LIN {X 0,Y 531.944,Z 396.877,A -85,B 0,C 180,E1 -4217.795,E2 -4217.795} C_VEL
LIN {X 0,Y 531.768,Z 407.802,A -85,B 0,C 180,E1 -4218.459,E2 -4218.459} C_VEL
LIN {X 0,Y 531.496,Z 419.072,A -85,B 0,C 180,E1 -4219.33,E2 -4219.33} C_VEL
LIN {X 0,Y 531.238,Z 429.006,A -85,B 0,C 180,E1 -4220.288,E2 -4220.288} C_VEL
LIN {X 0,Y 530.96,Z 438.48,A -85,B 0,C 180,E1 -4221.435,E2 -4221.435} C_VEL
LIN {X 0,Y 530.755,Z 446.079,A -85,B 0,C 180,E1 -4222.58,E2 -4222.58} C_VEL
LIN {X 0,Y 530.616,Z 451.92,A -85,B 0,C 180,E1 -4223.683,E2 -4223.683} C_VEL
LIN {X 0,Y 530.532,Z 456.21,A -85,B 0,C 180,E1 -4224.678,E2 -4224.678} C_VEL
LIN {X 0,Y 530.523,Z 460.056,A -85,B 0,C 180,E1 -4225.82,E2 -4225.82} C_VEL
LIN {X 0,Y 530.487,Z 462.909,A -85,B 0,C 180,E1 -4226.961,E2 -4226.961} C_VEL
LIN {X 0,Y 530.412,Z 464.34,A -85,B 0,C 180,E1 -4227.72,E2 -4227.72} C_VEL
LIN {X 0,Y 530.345,Z 465.895,A -85,B 0,C 180,E1 -4229.239,E2 -4229.239} C_VEL
LIN {X 0,Y 530.345,Z 466.145,A -85,B 0,C 180,E1 -4229.998,E2 -4229.998} C_VEL
LIN {X 0,Y 530.361,Z 465.393,A -85,B 0,C 180,E1 -4231.517,E2 -4231.517} C_VEL
LIN {X 0,Y 530.411,Z 464.474,A -85,B 0,C 180,E1 -4232.276,E2 -4232.276} C_VEL
LIN {X 0,Y 530.516,Z 461.35,A -85,B 0,C 180,E1 -4233.796,E2 -4233.796} C_VEL
LIN {X 0,Y 530.485,Z 457.917,A -85,B 0,C 180,E1 -4234.938,E2 -4234.938} C_VEL
LIN {X 0,Y 530.621,Z 453.388,A -85,B 0,C 180,E1 -4236.08,E2 -4236.08} C_VEL
LIN {X 0,Y 530.719,Z 447.667,A -85,B 0,C 180,E1 -4237.225,E2 -4237.225} C_VEL
LIN {X 0,Y 530.93,Z 440.518,A -85,B 0,C 180,E1 -4238.37,E2 -4238.37} C_VEL
LIN {X 0,Y 531.119,Z 433.212,A -85,B 0,C 180,E1 -4239.327,E2 -4239.327} C_VEL
LIN {X 0,Y 531.352,Z 423.28,A -85,B 0,C 180,E1 -4240.38,E2 -4240.38} C_VEL
LIN {X 0,Y 531.625,Z 413.173,A -85,B 0,C 180,E1 -4241.242,E2 -4241.242} C_VEL
LIN {X 0,Y 531.843,Z 401.662,A -85,B 0,C 180,E1 -4242.025,E2 -4242.025} C_VEL
LIN {X 0,Y 532.086,Z 388.922,A -85,B 0,C 180,E1 -4242.683,E2 -4242.683} C_VEL
LIN {X 0,Y 532.305,Z 376.104,A -85,B 0,C 180,E1 -4243.163,E2 -4243.163} C_VEL
LIN {X 0,Y 532.142,Z 370.063,A -85,B 0,C 180,E1 -4243.337,E2 -4243.337} C_VEL
LIN {X 0,Y 530.699,Z 362.74,A -85,B 0,C 180,E1 -4243.544,E2 -4243.544} C_VEL
LIN {X 0,Y 530.77,Z 357.319,A -85,B 0,C 180,E1 -4246.142,E2 -4246.142} C_VEL
LIN {X 0,Y 530.851,Z 352.311,A -85,B 0,C 180,E1 -4248.524,E2 -4248.524} C_VEL
LIN {X 0,Y 530.919,Z 347.179,A -85,B 0,C 180,E1 -4250.939,E2 -4250.939} C_VEL
LIN {X 0,Y 531.003,Z 340.698,A -85,B 0,C 180,E1 -4254.043,E2 -4254.043} C_VEL
LIN {X 0,Y 531.083,Z 335.26,A -85,B 0,C 180,E1 -4256.737,E2 -4256.737} C_VEL
LIN {X 0,Y 531.199,Z 330.065,A -85,B 0,C 180,E1 -4259.307,E2 -4259.307} C_VEL
LIN {X 0,Y 531.287,Z 323.918,A -85,B 0,C 180,E1 -4262.155,E2 -4262.155} C_VEL
LIN {X 0,Y 531.296,Z 317.258,A -85,B 0,C 180,E1 -4264.901,E2 -4264.901} C_VEL
LIN {X 0,Y 531.069,Z 314.65,A -85,B 0,C 180,E1 -4265.908,E2 -4265.908} C_VEL
LIN {X 0,Y 530.976,Z 314.657,A -85,B 0,C 180,E1 -4269.441,E2 -4269.441} C_VEL
LIN {X 0,Y 530.948,Z 314.659,A -85,B 0,C 180,E1 -4272.456,E2 -4272.456} C_VEL
LIN {X 0,Y 530.97,Z 314.657,A -85,B 0,C 180,E1 -4275.619,E2 -4275.619} C_VEL
LIN {X 0,Y 531.003,Z 314.656,A -85,B 0,C 180,E1 -4278.565,E2 -4278.565} C_VEL
LIN {X 0,Y 531.005,Z 314.656,A -85,B 0,C 180,E1 -4280.558,E2 -4280.558} C_VEL
LIN {X 0,Y 530.953,Z 314.663,A -85,B 0,C 180,E1 -4283.841,E2 -4283.841} C_VEL
LIN {X 0,Y 530.979,Z 314.653,A -85,B 0,C 180,E1 -4286.492,E2 -4286.492} C_VEL
LIN {X 0,Y 530.953,Z 314.66,A -85,B 0,C 180,E1 -4289.353,E2 -4289.353} C_VEL
LIN {X 0,Y 530.997,Z 314.656,A -85,B 0,C 180,E1 -4292.464,E2 -4292.464} C_VEL
LIN {X 0,Y 531,Z 314.652,A -85,B 0,C 180,E1 -4294.942,E2 -4294.942} C_VEL
LIN {X 0,Y 530.986,Z 314.657,A -85,B 0,C 180,E1 -4297.888,E2 -4297.888} C_VEL
LIN {X 0,Y 530.971,Z 314.654,A -85,B 0,C 180,E1 -4300.676,E2 -4300.676} C_VEL
LIN {X 0,Y 530.96,Z 314.662,A -85,B 0,C 180,E1 -4303.07,E2 -4303.07} C_VEL
LIN {X 0,Y 530.995,Z 314.649,A -85,B 0,C 180,E1 -4305.435,E2 -4305.435} C_VEL
LIN {X 0,Y 531.038,Z 314.65,A -85,B 0,C 180,E1 -4308.549,E2 -4308.549} C_VEL
LIN {X 0,Y 531.04,Z 314.647,A -85,B 0,C 180,E1 -4311.629,E2 -4311.629} C_VEL
LIN {X 0,Y 531.118,Z 314.635,A -85,B 0,C 180,E1 -4314.685,E2 -4314.685} C_VEL
LIN {X 0,Y 531.105,Z 314.639,A -85,B 0,C 180,E1 -4317.725,E2 -4317.725} C_VEL
LIN {X 0,Y 531.135,Z 314.637,A -85,B 0,C 180,E1 -4320.758,E2 -4320.758} C_VEL
LIN {X 0,Y 531.092,Z 314.64,A -85,B 0,C 180,E1 -4323.034,E2 -4323.034} C_VEL
LIN {X 0,Y 531.072,Z 314.646,A -85,B 0,C 180,E1 -4326.077,E2 -4326.077} C_VEL
LIN {X 0,Y 531.015,Z 314.654,A -85,B 0,C 180,E1 -4329.138,E2 -4329.138} C_VEL
LIN {X 0,Y 531.041,Z 314.647,A -85,B 0,C 180,E1 -4331.681,E2 -4331.681} C_VEL
LIN {X 0,Y 531.004,Z 314.653,A -85,B 0,C 180,E1 -4334.956,E2 -4334.956} C_VEL
LIN {X 0,Y 531.005,Z 314.653,A -85,B 0,C 180,E1 -4337.722,E2 -4337.722} C_VEL
LIN {X 0,Y 530.985,Z 314.654,A -85,B 0,C 180,E1 -4340.938,E2 -4340.938} C_VEL
LIN {X 0,Y 530.993,Z 314.652,A -85,B 0,C 180,E1 -4344.048,E2 -4344.048} C_VEL
LIN {X 0,Y 530.971,Z 314.66,A -85,B 0,C 180,E1 -4346.745,E2 -4346.745} C_VEL
LIN {X 0,Y 530.958,Z 314.656,A -85,B 0,C 180,E1 -4349.324,E2 -4349.324} C_VEL
LIN {X 0,Y 530.959,Z 314.663,A -85,B 0,C 180,E1 -4352.105,E2 -4352.105} C_VEL
LIN {X 0,Y 530.972,Z 314.656,A -85,B 0,C 180,E1 -4354.856,E2 -4354.856} C_VEL
LIN {X 0,Y 530.953,Z 314.661,A -85,B 0,C 180,E1 -4357.508,E2 -4357.508} C_VEL
LIN {X 0,Y 530.964,Z 314.658,A -85,B 0,C 180,E1 -4360.434,E2 -4360.434} C_VEL
LIN {X 0,Y 530.94,Z 314.658,A -85,B 0,C 180,E1 -4363.283,E2 -4363.283} C_VEL
LIN {X 0,Y 530.969,Z 314.659,A -85,B 0,C 180,E1 -4365.623,E2 -4365.623} C_VEL
LIN {X 0,Y 531.002,Z 314.655,A -85,B 0,C 180,E1 -4368.569,E2 -4368.569} C_VEL
LIN {X 0,Y 530.962,Z 314.677,A -85,B 0,C 180,E1 -4370.946,E2 -4370.946} C_VEL
LIN {X 0,Y 534.217,Z 325.862,A -85,B 0,C 180,E1 -4373.111,E2 -4373.111} C_VEL
LIN {X 0,Y 536.261,Z 334.019,A -85,B 0,C 180,E1 -4374.572,E2 -4374.572} C_VEL
LIN {X 0,Y 535.432,Z 353.193,A -85,B 0,C 180,E1 -4377.445,E2 -4377.445} C_VEL
LIN {X 0,Y 534.6,Z 374.419,A -85,B 0,C 180,E1 -4380.536,E2 -4380.536} C_VEL
LIN {X 0,Y 533.898,Z 393.207,A -85,B 0,C 180,E1 -4383.204,E2 -4383.204} C_VEL
LIN {X 0,Y 533.249,Z 412.473,A -85,B 0,C 180,E1 -4385.888,E2 -4385.888} C_VEL
LIN {X 0,Y 533.044,Z 420.982,A -85,B 0,C 180,E1 -4387.036,E2 -4387.036} C_VEL
LIN {X 0,Y 536.002,Z 434.729,A -85,B 0,C 180,E1 -4387.369,E2 -4387.369} C_VEL
LIN {X 0,Y 535.772,Z 451.721,A -85,B 0,C 180,E1 -4387.694,E2 -4387.694} C_VEL
LIN {X 0,Y 535.354,Z 468.564,A -85,B 0,C 180,E1 -4388.183,E2 -4388.183} C_VEL
LIN {X 0,Y 534.941,Z 483.544,A -85,B 0,C 180,E1 -4388.765,E2 -4388.765} C_VEL
LIN {X 0,Y 534.385,Z 498.799,A -85,B 0,C 180,E1 -4389.505,E2 -4389.505} C_VEL
LIN {X 0,Y 533.829,Z 513.607,A -85,B 0,C 180,E1 -4390.386,E2 -4390.386} C_VEL
LIN {X 0,Y 533.23,Z 528.49,A -85,B 0,C 180,E1 -4391.462,E2 -4391.462} C_VEL
LIN {X 0,Y 532.631,Z 542.063,A -85,B 0,C 180,E1 -4392.633,E2 -4392.633} C_VEL
LIN {X 0,Y 532.098,Z 554.523,A -85,B 0,C 180,E1 -4393.899,E2 -4393.899} C_VEL
LIN {X 0,Y 531.711,Z 566.234,A -85,B 0,C 180,E1 -4395.298,E2 -4395.298} C_VEL
LIN {X 0,Y 531.225,Z 576.99,A -85,B 0,C 180,E1 -4396.81,E2 -4396.81} C_VEL
LIN {X 0,Y 530.995,Z 586.264,A -85,B 0,C 180,E1 -4398.357,E2 -4398.357} C_VEL
LIN {X 0,Y 530.697,Z 594.864,A -85,B 0,C 180,E1 -4400.089,E2 -4400.089} C_VEL
LIN {X 0,Y 530.606,Z 601.058,A -85,B 0,C 180,E1 -4401.624,E2 -4401.624} C_VEL
LIN {X 0,Y 530.544,Z 606.129,A -85,B 0,C 180,E1 -4403.155,E2 -4403.155} C_VEL
LIN {X 0,Y 530.469,Z 610.061,A -85,B 0,C 180,E1 -4404.681,E2 -4404.681} C_VEL
LIN {X 0,Y 530.477,Z 612.984,A -85,B 0,C 180,E1 -4406.204,E2 -4406.204} C_VEL
LIN {X 0,Y 530.405,Z 614.894,A -85,B 0,C 180,E1 -4407.724,E2 -4407.724} C_VEL
LIN {X 0,Y 530.34,Z 615.85,A -85,B 0,C 180,E1 -4409.243,E2 -4409.243} C_VEL
LIN {X 0,Y 530.34,Z 615.849,A -85,B 0,C 180,E1 -4410.761,E2 -4410.761} C_VEL
LIN {X 0,Y 530.406,Z 614.891,A -85,B 0,C 180,E1 -4412.28,E2 -4412.28} C_VEL
LIN {X 0,Y 530.478,Z 612.978,A -85,B 0,C 180,E1 -4413.8,E2 -4413.8} C_VEL
LIN {X 0,Y 530.47,Z 610.055,A -85,B 0,C 180,E1 -4415.323,E2 -4415.323} C_VEL
LIN {X 0,Y 530.548,Z 606.119,A -85,B 0,C 180,E1 -4416.849,E2 -4416.849} C_VEL
LIN {X 0,Y 530.602,Z 601.043,A -85,B 0,C 180,E1 -4418.379,E2 -4418.379} C_VEL
LIN {X 0,Y 530.697,Z 594.849,A -85,B 0,C 180,E1 -4419.915,E2 -4419.915} C_VEL
LIN {X 0,Y 530.997,Z 586.255,A -85,B 0,C 180,E1 -4421.644,E2 -4421.644} C_VEL
LIN {X 0,Y 531.23,Z 576.964,A -85,B 0,C 180,E1 -4423.193,E2 -4423.193} C_VEL
LIN {X 0,Y 531.683,Z 566.209,A -85,B 0,C 180,E1 -4424.705,E2 -4424.705} C_VEL
LIN {X 0,Y 532.096,Z 554.492,A -85,B 0,C 180,E1 -4426.105,E2 -4426.105} C_VEL
LIN {X 0,Y 532.632,Z 542.024,A -85,B 0,C 180,E1 -4427.371,E2 -4427.371} C_VEL
LIN {X 0,Y 533.202,Z 528.444,A -85,B 0,C 180,E1 -4428.543,E2 -4428.543} C_VEL
LIN {X 0,Y 533.841,Z 513.547,A -85,B 0,C 180,E1 -4429.617,E2 -4429.617} C_VEL
LIN {X 0,Y 534.4,Z 498.726,A -85,B 0,C 180,E1 -4430.498,E2 -4430.498} C_VEL
LIN {X 0,Y 534.964,Z 483.415,A -85,B 0,C 180,E1 -4431.239,E2 -4431.239} C_VEL
LIN {X 0,Y 535.363,Z 468.451,A -85,B 0,C 180,E1 -4431.82,E2 -4431.82} C_VEL
LIN {X 0,Y 535.775,Z 451.557,A -85,B 0,C 180,E1 -4432.309,E2 -4432.309} C_VEL
LIN {X 0,Y 535.922,Z 433.878,A -85,B 0,C 180,E1 -4432.649,E2 -4432.649} C_VEL
LIN {X 0,Y 533.022,Z 420.656,A -85,B 0,C 180,E1 -4432.986,E2 -4432.986} C_VEL
LIN {X 0,Y 533.653,Z 400.588,A -85,B 0,C 180,E1 -4435.761,E2 -4435.761} C_VEL
LIN {X 0,Y 534.436,Z 378.358,A -85,B 0,C 180,E1 -4438.901,E2 -4438.901} C_VEL
LIN {X 0,Y 535.254,Z 357.61,A -85,B 0,C 180,E1 -4441.905,E2 -4441.905} C_VEL
LIN {X 0,Y 536.174,Z 336.862,A -85,B 0,C 180,E1 -4444.993,E2 -4444.993} C_VEL
LIN {X 0,Y 536.092,Z 332.802,A -85,B 0,C 180,E1 -4445.63,E2 -4445.63} C_VEL
LIN {X 0,Y 533.416,Z 322.296,A -85,B 0,C 180,E1 -4447.766,E2 -4447.766} C_VEL
LIN {X 0,Y 530.987,Z 314.659,A -85,B 0,C 180,E1 -4449.721,E2 -4449.721} C_VEL
LIN {X 0,Y 530.968,Z 314.66,A -85,B 0,C 180,E1 -4452.459,E2 -4452.459} C_VEL
LIN {X 0,Y 530.974,Z 314.66,A -85,B 0,C 180,E1 -4455.452,E2 -4455.452} C_VEL
LIN {X 0,Y 530.983,Z 314.66,A -85,B 0,C 180,E1 -4458.564,E2 -4458.564} C_VEL
LIN {X 0,Y 530.958,Z 314.663,A -85,B 0,C 180,E1 -4461.53,E2 -4461.53} C_VEL
LIN {X 0,Y 531.012,Z 314.81,A -85,B 0,C 180,E1 -4463.562,E2 -4463.562} C_VEL
LIN {X 0,Y 531.686,Z 319.123,A -85,B 0,C 180,E1 -4465.362,E2 -4465.362} C_VEL
LIN {X 0,Y 531.548,Z 325.536,A -85,B 0,C 180,E1 -4468.071,E2 -4468.071} C_VEL
LIN {X 0,Y 531.47,Z 331.546,A -85,B 0,C 180,E1 -4470.783,E2 -4470.783} C_VEL
LIN {X 0,Y 531.361,Z 336.706,A -85,B 0,C 180,E1 -4473.276,E2 -4473.276} C_VEL
LIN {X 0,Y 531.276,Z 341.953,A -85,B 0,C 180,E1 -4475.892,E2 -4475.892} C_VEL
LIN {X 0,Y 531.167,Z 346.592,A -85,B 0,C 180,E1 -4478.255,E2 -4478.255} C_VEL
LIN {X 0,Y 531.018,Z 351.305,A -85,B 0,C 180,E1 -4480.678,E2 -4480.678} C_VEL
LIN {X 0,Y 530.818,Z 355.833,A -85,B 0,C 180,E1 -4483.066,E2 -4483.066} C_VEL
LIN {X 0,Y 530.768,Z 360.402,A -85,B 0,C 180,E1 -4485.429,E2 -4485.429} C_VEL
LIN {X 0,Y 530.677,Z 362.403,A -85,B 0,C 180,E1 -4486.429,E2 -4486.429} C_VEL
LIN {X 0,Y 532.195,Z 368.999,A -85,B 0,C 180,E1 -4486.638,E2 -4486.638} C_VEL
LIN {X 0,Y 532.587,Z 374.814,A -85,B 0,C 180,E1 -4486.818,E2 -4486.818} C_VEL
LIN {X 0,Y 532.334,Z 387.141,A -85,B 0,C 180,E1 -4487.273,E2 -4487.273} C_VEL
LIN {X 0,Y 531.992,Z 399.267,A -85,B 0,C 180,E1 -4487.877,E2 -4487.877} C_VEL
LIN {X 0,Y 531.743,Z 411.267,A -85,B 0,C 180,E1 -4488.662,E2 -4488.662} C_VEL
LIN {X 0,Y 531.45,Z 421.692,A -85,B 0,C 180,E1 -4489.524,E2 -4489.524} C_VEL
LIN {X 0,Y 531.217,Z 431.074,A -85,B 0,C 180,E1 -4490.481,E2 -4490.481} C_VEL
LIN {X 0,Y 530.996,Z 438.766,A -85,B 0,C 180,E1 -4491.437,E2 -4491.437} C_VEL
LIN {X 0,Y 530.79,Z 446.287,A -85,B 0,C 180,E1 -4492.583,E2 -4492.583} C_VEL
LIN {X 0,Y 530.665,Z 453.159,A -85,B 0,C 180,E1 -4493.918,E2 -4493.918} C_VEL
LIN {X 0,Y 530.505,Z 457.747,A -85,B 0,C 180,E1 -4495.06,E2 -4495.06} C_VEL
LIN {X 0,Y 530.517,Z 461.232,A -85,B 0,C 180,E1 -4496.202,E2 -4496.202} C_VEL
LIN {X 0,Y 530.487,Z 463.037,A -85,B 0,C 180,E1 -4496.963,E2 -4496.963} C_VEL
LIN {X 0,Y 530.411,Z 464.41,A -85,B 0,C 180,E1 -4497.722,E2 -4497.722} C_VEL
LIN {X 0,Y 530.346,Z 465.975,A -85,B 0,C 180,E1 -4499.241,E2 -4499.241} C_VEL
LIN {X 0,Y 530.346,Z 466.196,A -85,B 0,C 180,E1 -4500,E2 -4500} C_VEL
LIN {X 0,Y 530.362,Z 465.438,A -85,B 0,C 180,E1 -4501.519,E2 -4501.519} C_VEL
LIN {X 0,Y 530.488,Z 463.149,A -85,B 0,C 180,E1 -4503.038,E2 -4503.038} C_VEL
LIN {X 0,Y 530.523,Z 460.342,A -85,B 0,C 180,E1 -4504.179,E2 -4504.179} C_VEL
LIN {X 0,Y 530.525,Z 456.536,A -85,B 0,C 180,E1 -4505.321,E2 -4505.321} C_VEL
LIN {X 0,Y 530.659,Z 450.689,A -85,B 0,C 180,E1 -4506.644,E2 -4506.644} C_VEL
LIN {X 0,Y 530.824,Z 444.156,A -85,B 0,C 180,E1 -4507.8,E2 -4507.8} C_VEL
LIN {X 0,Y 530.983,Z 436.105,A -85,B 0,C 180,E1 -4508.947,E2 -4508.947} C_VEL
LIN {X 0,Y 531.193,Z 427.816,A -85,B 0,C 180,E1 -4509.904,E2 -4509.904} C_VEL
LIN {X 0,Y 531.451,Z 417.592,A -85,B 0,C 180,E1 -4510.862,E2 -4510.862} C_VEL
LIN {X 0,Y 531.734,Z 405.832,A -85,B 0,C 180,E1 -4511.741,E2 -4511.741} C_VEL
LIN {X 0,Y 532.026,Z 394.618,A -85,B 0,C 180,E1 -4512.396,E2 -4512.396} C_VEL
LIN {X 0,Y 532.257,Z 381.529,A -85,B 0,C 180,E1 -4512.972,E2 -4512.972} C_VEL
LIN {X 0,Y 532.272,Z 370.626,A -85,B 0,C 180,E1 -4513.324,E2 -4513.324} C_VEL
LIN {X 0,Y 530.539,Z 361.418,A -85,B 0,C 180,E1 -4513.6,E2 -4513.6} C_VEL
LIN {X 0,Y 530.597,Z 356.022,A -85,B 0,C 180,E1 -4516.15,E2 -4516.15} C_VEL
LIN {X 0,Y 530.661,Z 351.011,A -85,B 0,C 180,E1 -4518.533,E2 -4518.533} C_VEL
LIN {X 0,Y 530.816,Z 344.274,A -85,B 0,C 180,E1 -4521.76,E2 -4521.76} C_VEL
LIN {X 0,Y 530.875,Z 337.416,A -85,B 0,C 180,E1 -4525.064,E2 -4525.064} C_VEL
LIN {X 0,Y 530.964,Z 332.154,A -85,B 0,C 180,E1 -4527.599,E2 -4527.599} C_VEL
LIN {X 0,Y 531.05,Z 325.866,A -85,B 0,C 180,E1 -4530.657,E2 -4530.657} C_VEL
LIN {X 0,Y 531.166,Z 319.995,A -85,B 0,C 180,E1 -4533.531,E2 -4533.531} C_VEL
LIN {X 0,Y 531.105,Z 315.782,A -85,B 0,C 180,E1 -4535.609,E2 -4535.609} C_VEL
LIN {X 0,Y 531.013,Z 314.656,A -85,B 0,C 180,E1 -4536.212,E2 -4536.212} C_VEL
LIN {X 0,Y 530.948,Z 314.662,A -85,B 0,C 180,E1 -4537.998,E2 -4537.998} C_VEL
LIN {X 0,Y 530.295,Z 314.746,A -85,B 0,C 180,E1 -4538.632,E2 -4538.632} C_VEL
LIN {X 0,Y 527.485,Z 315.099,A -85,B 0,C 180,E1 -4539.661,E2 -4539.661} C_VEL
LIN {X 0,Y 525.096,Z 315.398,A -85,B 0,C 180,E1 -4540.49,E2 -4540.49} C_VEL
LIN {X 0,Y 524.052,Z 315.525,A -85,B 0,C 180,E1 -4541.129,E2 -4541.129} C_VEL
LIN {X 0,Y 523.958,Z 315.534,A -85,B 0,C 180,E1 -4541.345,E2 -4541.345} C_VEL
LIN {X 0,Y 523.949,Z 315.532,A -85,B 0,C 180,E1 -4544.689,E2 -4544.689} C_VEL
LIN {X 0,Y 523.948,Z 315.535,A -85,B 0,C 180,E1 -4547.879,E2 -4547.879} C_VEL
LIN {X 0,Y 523.921,Z 315.537,A -85,B 0,C 180,E1 -4550.914,E2 -4550.914} C_VEL
LIN {X 0,Y 523.978,Z 315.637,A -85,B 0,C 180,E1 -4554.127,E2 -4554.127} C_VEL
LIN {X 0,Y 524.311,Z 320.951,A -85,B 0,C 180,E1 -4556.209,E2 -4556.209} C_VEL
LIN {X 0,Y 524.237,Z 327.536,A -85,B 0,C 180,E1 -4559.093,E2 -4559.093} C_VEL
LIN {X 0,Y 524.146,Z 331.854,A -85,B 0,C 180,E1 -4561.136,E2 -4561.136} C_VEL
LIN {X 0,Y 524.062,Z 337.559,A -85,B 0,C 180,E1 -4563.964,E2 -4563.964} C_VEL
LIN {X 0,Y 523.929,Z 343.888,A -85,B 0,C 180,E1 -4567.106,E2 -4567.106} C_VEL
LIN {X 0,Y 523.87,Z 349.762,A -85,B 0,C 180,E1 -4569.9,E2 -4569.9} C_VEL
LIN {X 0,Y 523.795,Z 356.084,A -85,B 0,C 180,E1 -4572.83,E2 -4572.83} C_VEL
LIN {X 0,Y 523.794,Z 361.232,A -85,B 0,C 180,E1 -4575.229,E2 -4575.229} C_VEL
LIN {X 0,Y 523.761,Z 363.654,A -85,B 0,C 180,E1 -4576.368,E2 -4576.368} C_VEL
LIN {X 0,Y 525.52,Z 372.2,A -85,B 0,C 180,E1 -4576.611,E2 -4576.611} C_VEL
LIN {X 0,Y 525.333,Z 385.421,A -85,B 0,C 180,E1 -4577.049,E2 -4577.049} C_VEL
LIN {X 0,Y 525.078,Z 397.932,A -85,B 0,C 180,E1 -4577.632,E2 -4577.632} C_VEL
LIN {X 0,Y 524.898,Z 408.921,A -85,B 0,C 180,E1 -4578.31,E2 -4578.31} C_VEL
LIN {X 0,Y 524.611,Z 420.135,A -85,B 0,C 180,E1 -4579.188,E2 -4579.188} C_VEL
LIN {X 0,Y 524.339,Z 430.071,A -85,B 0,C 180,E1 -4580.158,E2 -4580.158} C_VEL
LIN {X 0,Y 524.046,Z 439.543,A -85,B 0,C 180,E1 -4581.321,E2 -4581.321} C_VEL
LIN {X 0,Y 523.802,Z 447.15,A -85,B 0,C 180,E1 -4582.481,E2 -4582.481} C_VEL
LIN {X 0,Y 523.655,Z 453.221,A -85,B 0,C 180,E1 -4583.644,E2 -4583.644} C_VEL
LIN {X 0,Y 523.498,Z 458.684,A -85,B 0,C 180,E1 -4584.992,E2 -4584.992} C_VEL
LIN {X 0,Y 523.517,Z 462.195,A -85,B 0,C 180,E1 -4586.149,E2 -4586.149} C_VEL
LIN {X 0,Y 523.482,Z 464.009,A -85,B 0,C 180,E1 -4586.92,E2 -4586.92} C_VEL
LIN {X 0,Y 523.42,Z 465.405,A -85,B 0,C 180,E1 -4587.69,E2 -4587.69} C_VEL
LIN {X 0,Y 523.355,Z 466.985,A -85,B 0,C 180,E1 -4589.229,E2 -4589.229} C_VEL
LIN {X 0,Y 523.351,Z 467.219,A -85,B 0,C 180,E1 -4589.998,E2 -4589.998} C_VEL
LIN {X 0,Y 523.355,Z 466.477,A -85,B 0,C 180,E1 -4591.537,E2 -4591.537} C_VEL
LIN {X 0,Y 523.511,Z 464.205,A -85,B 0,C 180,E1 -4593.076,E2 -4593.076} C_VEL
LIN {X 0,Y 523.539,Z 461.425,A -85,B 0,C 180,E1 -4594.232,E2 -4594.232} C_VEL
LIN {X 0,Y 523.562,Z 457.648,A -85,B 0,C 180,E1 -4595.39,E2 -4595.39} C_VEL
LIN {X 0,Y 523.679,Z 451.858,A -85,B 0,C 180,E1 -4596.726,E2 -4596.726} C_VEL
LIN {X 0,Y 523.873,Z 445.359,A -85,B 0,C 180,E1 -4597.902,E2 -4597.902} C_VEL
LIN {X 0,Y 524.116,Z 437.372,A -85,B 0,C 180,E1 -4599.063,E2 -4599.063} C_VEL
LIN {X 0,Y 524.348,Z 429.129,A -85,B 0,C 180,E1 -4600.032,E2 -4600.032} C_VEL
LIN {X 0,Y 524.627,Z 418.982,A -85,B 0,C 180,E1 -4601.003,E2 -4601.003} C_VEL
LIN {X 0,Y 524.89,Z 409.008,A -85,B 0,C 180,E1 -4601.774,E2 -4601.774} C_VEL
LIN {X 0,Y 525.105,Z 397.849,A -85,B 0,C 180,E1 -4602.461,E2 -4602.461} C_VEL
LIN {X 0,Y 525.357,Z 385.312,A -85,B 0,C 180,E1 -4603.045,E2 -4603.045} C_VEL
LIN {X 0,Y 525.513,Z 372.944,A -85,B 0,C 180,E1 -4603.459,E2 -4603.459} C_VEL
LIN {X 0,Y 524.183,Z 365.367,A -85,B 0,C 180,E1 -4603.675,E2 -4603.675} C_VEL
LIN {X 0,Y 523.75,Z 363.666,A -85,B 0,C 180,E1 -4603.728,E2 -4603.728} C_VEL
LIN {X 0,Y 523.768,Z 358.003,A -85,B 0,C 180,E1 -4606.364,E2 -4606.364} C_VEL
LIN {X 0,Y 523.83,Z 352.816,A -85,B 0,C 180,E1 -4608.781,E2 -4608.781} C_VEL
LIN {X 0,Y 523.889,Z 347.557,A -85,B 0,C 180,E1 -4611.233,E2 -4611.233} C_VEL
LIN {X 0,Y 523.999,Z 341.39,A -85,B 0,C 180,E1 -4614.211,E2 -4614.211} C_VEL
LIN {X 0,Y 524.083,Z 335.577,A -85,B 0,C 180,E1 -4617.123,E2 -4617.123} C_VEL
LIN {X 0,Y 524.199,Z 330.259,A -85,B 0,C 180,E1 -4619.737,E2 -4619.737} C_VEL
LIN {X 0,Y 524.262,Z 324.408,A -85,B 0,C 180,E1 -4622.424,E2 -4622.424} C_VEL
LIN {X 0,Y 524.27,Z 318.925,A -85,B 0,C 180,E1 -4624.699,E2 -4624.699} C_VEL
LIN {X 0,Y 523.994,Z 315.531,A -85,B 0,C 180,E1 -4626.045,E2 -4626.045} C_VEL
LIN {X 0,Y 523.91,Z 315.536,A -85,B 0,C 180,E1 -4629.082,E2 -4629.082} C_VEL
LIN {X 0,Y 523.925,Z 315.535,A -85,B 0,C 180,E1 -4632.118,E2 -4632.118} C_VEL
LIN {X 0,Y 523.936,Z 315.536,A -85,B 0,C 180,E1 -4635.307,E2 -4635.307} C_VEL
LIN {X 0,Y 523.966,Z 315.535,A -85,B 0,C 180,E1 -4638.684,E2 -4638.684} C_VEL
LIN {X 0,Y 523.941,Z 315.531,A -85,B 0,C 180,E1 -4641.073,E2 -4641.073} C_VEL
LIN {X 0,Y 523.908,Z 315.541,A -85,B 0,C 180,E1 -4643.825,E2 -4643.825} C_VEL
LIN {X 0,Y 523.921,Z 315.533,A -85,B 0,C 180,E1 -4646.634,E2 -4646.634} C_VEL
LIN {X 0,Y 523.934,Z 315.534,A -85,B 0,C 180,E1 -4649.354,E2 -4649.354} C_VEL
LIN {X 0,Y 523.959,Z 315.531,A -85,B 0,C 180,E1 -4652.279,E2 -4652.279} C_VEL
LIN {X 0,Y 523.943,Z 315.535,A -85,B 0,C 180,E1 -4654.58,E2 -4654.58} C_VEL
LIN {X 0,Y 523.942,Z 315.528,A -85,B 0,C 180,E1 -4657.108,E2 -4657.108} C_VEL
LIN {X 0,Y 523.956,Z 315.531,A -85,B 0,C 180,E1 -4659.864,E2 -4659.864} C_VEL
LIN {X 0,Y 523.942,Z 315.533,A -85,B 0,C 180,E1 -4662.836,E2 -4662.836} C_VEL
LIN {X 0,Y 523.952,Z 315.528,A -85,B 0,C 180,E1 -4665.235,E2 -4665.235} C_VEL
LIN {X 0,Y 524.015,Z 315.528,A -85,B 0,C 180,E1 -4668.394,E2 -4668.394} C_VEL
LIN {X 0,Y 523.987,Z 315.524,A -85,B 0,C 180,E1 -4671.515,E2 -4671.515} C_VEL
LIN {X 0,Y 524.076,Z 315.512,A -85,B 0,C 180,E1 -4674.613,E2 -4674.613} C_VEL
LIN {X 0,Y 524.078,Z 315.514,A -85,B 0,C 180,E1 -4677.694,E2 -4677.694} C_VEL
LIN {X 0,Y 524.104,Z 315.512,A -85,B 0,C 180,E1 -4680.768,E2 -4680.768} C_VEL
LIN {X 0,Y 524.058,Z 315.516,A -85,B 0,C 180,E1 -4683.075,E2 -4683.075} C_VEL
LIN {X 0,Y 524.032,Z 315.522,A -85,B 0,C 180,E1 -4686.159,E2 -4686.159} C_VEL
LIN {X 0,Y 523.983,Z 315.531,A -85,B 0,C 180,E1 -4689.262,E2 -4689.262} C_VEL
LIN {X 0,Y 523.998,Z 315.524,A -85,B 0,C 180,E1 -4691.752,E2 -4691.752} C_VEL
LIN {X 0,Y 523.967,Z 315.529,A -85,B 0,C 180,E1 -4695.053,E2 -4695.053} C_VEL
LIN {X 0,Y 523.947,Z 315.536,A -85,B 0,C 180,E1 -4697.969,E2 -4697.969} C_VEL
LIN {X 0,Y 523.95,Z 315.53,A -85,B 0,C 180,E1 -4700.411,E2 -4700.411} C_VEL
LIN {X 0,Y 523.936,Z 315.533,A -85,B 0,C 180,E1 -4702.892,E2 -4702.892} C_VEL
LIN {X 0,Y 523.925,Z 315.535,A -85,B 0,C 180,E1 -4705.42,E2 -4705.42} C_VEL
LIN {X 0,Y 523.941,Z 315.531,A -85,B 0,C 180,E1 -4708,E2 -4708} C_VEL
LIN {X 0,Y 523.924,Z 315.534,A -85,B 0,C 180,E1 -4710.857,E2 -4710.857} C_VEL
LIN {X 0,Y 523.941,Z 315.537,A -85,B 0,C 180,E1 -4713.737,E2 -4713.737} C_VEL
LIN {X 0,Y 523.905,Z 315.536,A -85,B 0,C 180,E1 -4716.406,E2 -4716.406} C_VEL
LIN {X 0,Y 523.904,Z 315.54,A -85,B 0,C 180,E1 -4719.086,E2 -4719.086} C_VEL
LIN {X 0,Y 523.932,Z 315.532,A -85,B 0,C 180,E1 -4722.121,E2 -4722.121} C_VEL
LIN {X 0,Y 523.937,Z 315.534,A -85,B 0,C 180,E1 -4725.31,E2 -4725.31} C_VEL
LIN {X 0,Y 523.965,Z 315.532,A -85,B 0,C 180,E1 -4728.688,E2 -4728.688} C_VEL
LIN {X 0,Y 523.964,Z 315.654,A -85,B 0,C 180,E1 -4730.45,E2 -4730.45} C_VEL
LIN {X 0,Y 527.769,Z 328.728,A -85,B 0,C 180,E1 -4733.033,E2 -4733.033} C_VEL
LIN {X 0,Y 529.572,Z 335.49,A -85,B 0,C 180,E1 -4734.276,E2 -4734.276} C_VEL
LIN {X 0,Y 529.469,Z 341.343,A -85,B 0,C 180,E1 -4735.199,E2 -4735.199} C_VEL
LIN {X 0,Y 528.506,Z 361.199,A -85,B 0,C 180,E1 -4738.183,E2 -4738.183} C_VEL
LIN {X 0,Y 527.658,Z 381.351,A -85,B 0,C 180,E1 -4741.133,E2 -4741.133} C_VEL
LIN {X 0,Y 526.874,Z 400.617,A -85,B 0,C 180,E1 -4743.887,E2 -4743.887} C_VEL
LIN {X 0,Y 526.291,Z 418.401,A -85,B 0,C 180,E1 -4746.386,E2 -4746.386} C_VEL
LIN {X 0,Y 526.183,Z 420.755,A -85,B 0,C 180,E1 -4746.712,E2 -4746.712} C_VEL
LIN {X 0,Y 529.422,Z 435.739,A -85,B 0,C 180,E1 -4747.089,E2 -4747.089} C_VEL
LIN {X 0,Y 529.201,Z 452.269,A -85,B 0,C 180,E1 -4747.416,E2 -4747.416} C_VEL
LIN {X 0,Y 528.769,Z 468.565,A -85,B 0,C 180,E1 -4747.897,E2 -4747.897} C_VEL
LIN {X 0,Y 528.332,Z 482.558,A -85,B 0,C 180,E1 -4748.442,E2 -4748.442} C_VEL
LIN {X 0,Y 527.815,Z 497.033,A -85,B 0,C 180,E1 -4749.136,E2 -4749.136} C_VEL
LIN {X 0,Y 527.228,Z 510.493,A -85,B 0,C 180,E1 -4749.927,E2 -4749.927} C_VEL
LIN {X 0,Y 526.586,Z 524.647,A -85,B 0,C 180,E1 -4750.917,E2 -4750.917} C_VEL
LIN {X 0,Y 526,Z 537.537,A -85,B 0,C 180,E1 -4751.979,E2 -4751.979} C_VEL
LIN {X 0,Y 525.34,Z 550.962,A -85,B 0,C 180,E1 -4753.286,E2 -4753.286} C_VEL
LIN {X 0,Y 524.785,Z 563.745,A -85,B 0,C 180,E1 -4754.769,E2 -4754.769} C_VEL
LIN {X 0,Y 524.358,Z 574.421,A -85,B 0,C 180,E1 -4756.239,E2 -4756.239} C_VEL
LIN {X 0,Y 524.003,Z 584.177,A -85,B 0,C 180,E1 -4757.827,E2 -4757.827} C_VEL
LIN {X 0,Y 523.726,Z 593.063,A -85,B 0,C 180,E1 -4759.565,E2 -4759.565} C_VEL
LIN {X 0,Y 523.559,Z 599.635,A -85,B 0,C 180,E1 -4761.122,E2 -4761.122} C_VEL
LIN {X 0,Y 523.467,Z 604.962,A -85,B 0,C 180,E1 -4762.674,E2 -4762.674} C_VEL
LIN {X 0,Y 523.41,Z 608.25,A -85,B 0,C 180,E1 -4763.835,E2 -4763.835} C_VEL
LIN {X 0,Y 523.311,Z 611.638,A -85,B 0,C 180,E1 -4765.38,E2 -4765.38} C_VEL
LIN {X 0,Y 523.353,Z 614.091,A -85,B 0,C 180,E1 -4766.923,E2 -4766.923} C_VEL
LIN {X 0,Y 523.268,Z 615.48,A -85,B 0,C 180,E1 -4768.463,E2 -4768.463} C_VEL
LIN {X 0,Y 523.242,Z 616,A -85,B 0,C 180,E1 -4770.002,E2 -4770.002} C_VEL
LIN {X 0,Y 523.269,Z 615.479,A -85,B 0,C 180,E1 -4771.541,E2 -4771.541} C_VEL
LIN {X 0,Y 523.354,Z 614.086,A -85,B 0,C 180,E1 -4773.081,E2 -4773.081} C_VEL
LIN {X 0,Y 523.312,Z 611.632,A -85,B 0,C 180,E1 -4774.624,E2 -4774.624} C_VEL
LIN {X 0,Y 523.412,Z 608.245,A -85,B 0,C 180,E1 -4776.168,E2 -4776.168} C_VEL
LIN {X 0,Y 523.471,Z 603.713,A -85,B 0,C 180,E1 -4777.717,E2 -4777.717} C_VEL
LIN {X 0,Y 523.564,Z 598.096,A -85,B 0,C 180,E1 -4779.271,E2 -4779.271} C_VEL
LIN {X 0,Y 523.788,Z 591.226,A -85,B 0,C 180,E1 -4780.829,E2 -4780.829} C_VEL
LIN {X 0,Y 524.039,Z 582.925,A -85,B 0,C 180,E1 -4782.392,E2 -4782.392} C_VEL
LIN {X 0,Y 524.378,Z 573.044,A -85,B 0,C 180,E1 -4783.962,E2 -4783.962} C_VEL
LIN {X 0,Y 524.802,Z 562.551,A -85,B 0,C 180,E1 -4785.378,E2 -4785.378} C_VEL
LIN {X 0,Y 525.345,Z 550.924,A -85,B 0,C 180,E1 -4786.717,E2 -4786.717} C_VEL
LIN {X 0,Y 525.973,Z 537.46,A -85,B 0,C 180,E1 -4788.028,E2 -4788.028} C_VEL
LIN {X 0,Y 526.631,Z 523.306,A -85,B 0,C 180,E1 -4789.187,E2 -4789.187} C_VEL
LIN {X 0,Y 527.294,Z 508.855,A -85,B 0,C 180,E1 -4790.176,E2 -4790.176} C_VEL
LIN {X 0,Y 527.876,Z 495.023,A -85,B 0,C 180,E1 -4790.967,E2 -4790.967} C_VEL
LIN {X 0,Y 528.428,Z 478.729,A -85,B 0,C 180,E1 -4791.725,E2 -4791.725} C_VEL
LIN {X 0,Y 528.94,Z 461.848,A -85,B 0,C 180,E1 -4792.322,E2 -4792.322} C_VEL
LIN {X 0,Y 529.309,Z 445.853,A -85,B 0,C 180,E1 -4792.726,E2 -4792.726} C_VEL
LIN {X 0,Y 529.299,Z 434.652,A -85,B 0,C 180,E1 -4792.936,E2 -4792.936} C_VEL
LIN {X 0,Y 526.166,Z 420.721,A -85,B 0,C 180,E1 -4793.293,E2 -4793.293} C_VEL
LIN {X 0,Y 526.855,Z 402.07,A -85,B 0,C 180,E1 -4795.906,E2 -4795.906} C_VEL
LIN {X 0,Y 527.631,Z 381.322,A -85,B 0,C 180,E1 -4798.873,E2 -4798.873} C_VEL
LIN {X 0,Y 528.577,Z 360.131,A -85,B 0,C 180,E1 -4801.974,E2 -4801.974} C_VEL
LIN {X 0,Y 529.547,Z 339.872,A -85,B 0,C 180,E1 -4805.031,E2 -4805.031} C_VEL
LIN {X 0,Y 529.597,Z 335.53,A -85,B 0,C 180,E1 -4805.727,E2 -4805.727} C_VEL
LIN {X 0,Y 527.136,Z 325.532,A -85,B 0,C 180,E1 -4807.829,E2 -4807.829} C_VEL
LIN {X 0,Y 524.849,Z 318.451,A -85,B 0,C 180,E1 -4809.651,E2 -4809.651} C_VEL
LIN {X 0,Y 523.944,Z 315.537,A -85,B 0,C 180,E1 -4810.585,E2 -4810.585} C_VEL
LIN {X 0,Y 523.914,Z 315.539,A -85,B 0,C 180,E1 -4813.583,E2 -4813.583} C_VEL
LIN {X 0,Y 523.908,Z 315.54,A -85,B 0,C 180,E1 -4816.419,E2 -4816.419} C_VEL
LIN {X 0,Y 523.922,Z 315.539,A -85,B 0,C 180,E1 -4818.906,E2 -4818.906} C_VEL
LIN {X 0,Y 523.918,Z 315.539,A -85,B 0,C 180,E1 -4821.899,E2 -4821.899} C_VEL
LIN {X 0,Y 523.962,Z 315.757,A -85,B 0,C 180,E1 -4823.068,E2 -4823.068} C_VEL
LIN {X 0,Y 524.731,Z 319.717,A -85,B 0,C 180,E1 -4824.836,E2 -4824.836} C_VEL
LIN {X 0,Y 524.748,Z 324.019,A -85,B 0,C 180,E1 -4826.694,E2 -4826.694} C_VEL
LIN {X 0,Y 524.607,Z 330.077,A -85,B 0,C 180,E1 -4829.398,E2 -4829.398} C_VEL
LIN {X 0,Y 524.483,Z 335.945,A -85,B 0,C 180,E1 -4832.178,E2 -4832.178} C_VEL
LIN {X 0,Y 524.347,Z 340.806,A -85,B 0,C 180,E1 -4834.602,E2 -4834.602} C_VEL
LIN {X 0,Y 524.224,Z 345.769,A -85,B 0,C 180,E1 -4837.121,E2 -4837.121} C_VEL
LIN {X 0,Y 524.079,Z 351.027,A -85,B 0,C 180,E1 -4839.839,E2 -4839.839} C_VEL
LIN {X 0,Y 523.87,Z 356.819,A -85,B 0,C 180,E1 -4842.834,E2 -4842.834} C_VEL
LIN {X 0,Y 523.818,Z 361.416,A -85,B 0,C 180,E1 -4845.231,E2 -4845.231} C_VEL
LIN {X 0,Y 523.756,Z 363.405,A -85,B 0,C 180,E1 -4846.197,E2 -4846.197} C_VEL
LIN {X 0,Y 525.351,Z 369.393,A -85,B 0,C 180,E1 -4846.397,E2 -4846.397} C_VEL
LIN {X 0,Y 525.853,Z 374.861,A -85,B 0,C 180,E1 -4846.573,E2 -4846.573} C_VEL
LIN {X 0,Y 525.582,Z 387.911,A -85,B 0,C 180,E1 -4847.058,E2 -4847.058} C_VEL
LIN {X 0,Y 525.194,Z 400.184,A -85,B 0,C 180,E1 -4847.678,E2 -4847.678} C_VEL
LIN {X 0,Y 524.948,Z 411.419,A -85,B 0,C 180,E1 -4848.415,E2 -4848.415} C_VEL
LIN {X 0,Y 524.625,Z 422.022,A -85,B 0,C 180,E1 -4849.288,E2 -4849.288} C_VEL
LIN {X 0,Y 524.365,Z 432.395,A -85,B 0,C 180,E1 -4850.356,E2 -4850.356} C_VEL
LIN {X 0,Y 524.113,Z 440.067,A -85,B 0,C 180,E1 -4851.324,E2 -4851.324} C_VEL
LIN {X 0,Y 523.894,Z 447.569,A -85,B 0,C 180,E1 -4852.485,E2 -4852.485} C_VEL
LIN {X 0,Y 523.719,Z 454.436,A -85,B 0,C 180,E1 -4853.837,E2 -4853.837} C_VEL
LIN {X 0,Y 523.551,Z 459.012,A -85,B 0,C 180,E1 -4854.995,E2 -4854.995} C_VEL
LIN {X 0,Y 523.572,Z 462.482,A -85,B 0,C 180,E1 -4856.152,E2 -4856.152} C_VEL
LIN {X 0,Y 523.512,Z 464.276,A -85,B 0,C 180,E1 -4856.922,E2 -4856.922} C_VEL
LIN {X 0,Y 523.447,Z 465.637,A -85,B 0,C 180,E1 -4857.692,E2 -4857.692} C_VEL
LIN {X 0,Y 523.356,Z 467.184,A -85,B 0,C 180,E1 -4859.231,E2 -4859.231} C_VEL
LIN {X 0,Y 523.352,Z 467.379,A -85,B 0,C 180,E1 -4860,E2 -4860} C_VEL
LIN {X 0,Y 523.382,Z 466.586,A -85,B 0,C 180,E1 -4861.539,E2 -4861.539} C_VEL
LIN {X 0,Y 523.419,Z 465.623,A -85,B 0,C 180,E1 -4862.309,E2 -4862.309} C_VEL
LIN {X 0,Y 523.483,Z 464.247,A -85,B 0,C 180,E1 -4863.079,E2 -4863.079} C_VEL
LIN {X 0,Y 523.522,Z 461.405,A -85,B 0,C 180,E1 -4864.235,E2 -4864.235} C_VEL
LIN {X 0,Y 523.538,Z 457.557,A -85,B 0,C 180,E1 -4865.392,E2 -4865.392} C_VEL
LIN {X 0,Y 523.69,Z 451.65,A -85,B 0,C 180,E1 -4866.734,E2 -4866.734} C_VEL
LIN {X 0,Y 523.868,Z 445.083,A -85,B 0,C 180,E1 -4867.904,E2 -4867.904} C_VEL
LIN {X 0,Y 524.051,Z 436.98,A -85,B 0,C 180,E1 -4869.067,E2 -4869.067} C_VEL
LIN {X 0,Y 524.257,Z 428.649,A -85,B 0,C 180,E1 -4870.037,E2 -4870.037} C_VEL
LIN {X 0,Y 524.553,Z 418.398,A -85,B 0,C 180,E1 -4871.007,E2 -4871.007} C_VEL
LIN {X 0,Y 524.838,Z 406.812,A -85,B 0,C 180,E1 -4871.884,E2 -4871.884} C_VEL
LIN {X 0,Y 525.155,Z 395.432,A -85,B 0,C 180,E1 -4872.561,E2 -4872.561} C_VEL
LIN {X 0,Y 525.379,Z 382.434,A -85,B 0,C 180,E1 -4873.145,E2 -4873.145} C_VEL
LIN {X 0,Y 525.371,Z 371.275,A -85,B 0,C 180,E1 -4873.514,E2 -4873.514} C_VEL
LIN {X 0,Y 523.482,Z 361.785,A -85,B 0,C 180,E1 -4873.811,E2 -4873.811} C_VEL
LIN {X 0,Y 523.553,Z 356.382,A -85,B 0,C 180,E1 -4876.374,E2 -4876.374} C_VEL
LIN {X 0,Y 523.608,Z 351.339,A -85,B 0,C 180,E1 -4878.792,E2 -4878.792} C_VEL
LIN {X 0,Y 523.792,Z 344.539,A -85,B 0,C 180,E1 -4882.067,E2 -4882.067} C_VEL
LIN {X 0,Y 523.832,Z 339.335,A -85,B 0,C 180,E1 -4884.577,E2 -4884.577} C_VEL
LIN {X 0,Y 523.943,Z 332.88,A -85,B 0,C 180,E1 -4887.71,E2 -4887.71} C_VEL
LIN {X 0,Y 524.029,Z 326.914,A -85,B 0,C 180,E1 -4890.64,E2 -4890.64} C_VEL
LIN {X 0,Y 524.145,Z 320.584,A -85,B 0,C 180,E1 -4893.763,E2 -4893.763} C_VEL
LIN {X 0,Y 523.987,Z 315.556,A -85,B 0,C 180,E1 -4896.277,E2 -4896.277} C_VEL
LIN {X 0,Y 523.92,Z 315.54,A -85,B 0,C 180,E1 -4899.085,E2 -4899.085} C_VEL
LIN {X 0,Y 523.958,Z 315.534,A -85,B 0,C 180,E1 -4901.345,E2 -4901.345} C_VEL
LIN {X 0,Y 523.259,Z 315.62,A -85,B 0,C 180,E1 -4901.986,E2 -4901.986} C_VEL
LIN {X 0,Y 520.371,Z 315.979,A -85,B 0,C 180,E1 -4903.025,E2 -4903.025} C_VEL
LIN {X 0,Y 517.963,Z 316.281,A -85,B 0,C 180,E1 -4903.862,E2 -4903.862} C_VEL
LIN {X 0,Y 516.953,Z 316.403,A -85,B 0,C 180,E1 -4904.509,E2 -4904.509} C_VEL
LIN {X 0,Y 516.883,Z 316.412,A -85,B 0,C 180,E1 -4904.728,E2 -4904.728} C_VEL
LIN {X 0,Y 516.866,Z 316.416,A -85,B 0,C 180,E1 -4907.245,E2 -4907.245} C_VEL
LIN {X 0,Y 516.893,Z 316.412,A -85,B 0,C 180,E1 -4909.589,E2 -4909.589} C_VEL
LIN {X 0,Y 516.869,Z 316.417,A -85,B 0,C 180,E1 -4912.273,E2 -4912.273} C_VEL
LIN {X 0,Y 516.92,Z 316.42,A -85,B 0,C 180,E1 -4913.982,E2 -4913.982} C_VEL
LIN {X 0,Y 517.31,Z 321.494,A -85,B 0,C 180,E1 -4915.969,E2 -4915.969} C_VEL
LIN {X 0,Y 517.232,Z 328.234,A -85,B 0,C 180,E1 -4918.912,E2 -4918.912} C_VEL
LIN {X 0,Y 517.099,Z 333.92,A -85,B 0,C 180,E1 -4921.594,E2 -4921.594} C_VEL
LIN {X 0,Y 517.013,Z 339.15,A -85,B 0,C 180,E1 -4924.214,E2 -4924.214} C_VEL
LIN {X 0,Y 516.922,Z 344.262,A -85,B 0,C 180,E1 -4926.777,E2 -4926.777} C_VEL
LIN {X 0,Y 516.853,Z 350.45,A -85,B 0,C 180,E1 -4929.759,E2 -4929.759} C_VEL
LIN {X 0,Y 516.8,Z 356.611,A -85,B 0,C 180,E1 -4932.59,E2 -4932.59} C_VEL
LIN {X 0,Y 516.764,Z 363.802,A -85,B 0,C 180,E1 -4935.828,E2 -4935.828} C_VEL
LIN {X 0,Y 516.796,Z 364.577,A -85,B 0,C 180,E1 -4936.181,E2 -4936.181} C_VEL
LIN {X 0,Y 518.527,Z 372.242,A -85,B 0,C 180,E1 -4936.402,E2 -4936.402} C_VEL
LIN {X 0,Y 518.544,Z 384.003,A -85,B 0,C 180,E1 -4936.777,E2 -4936.777} C_VEL
LIN {X 0,Y 518.306,Z 395.246,A -85,B 0,C 180,E1 -4937.269,E2 -4937.269} C_VEL
LIN {X 0,Y 518.066,Z 406.875,A -85,B 0,C 180,E1 -4937.943,E2 -4937.943} C_VEL
LIN {X 0,Y 517.82,Z 417.782,A -85,B 0,C 180,E1 -4938.748,E2 -4938.748} C_VEL
LIN {X 0,Y 517.523,Z 427.432,A -85,B 0,C 180,E1 -4939.632,E2 -4939.632} C_VEL
LIN {X 0,Y 517.29,Z 436.136,A -85,B 0,C 180,E1 -4940.615,E2 -4940.615} C_VEL
LIN {X 0,Y 516.983,Z 444.626,A -85,B 0,C 180,E1 -4941.792,E2 -4941.792} C_VEL
LIN {X 0,Y 516.779,Z 451.426,A -85,B 0,C 180,E1 -4942.968,E2 -4942.968} C_VEL
LIN {X 0,Y 516.68,Z 456.815,A -85,B 0,C 180,E1 -4944.143,E2 -4944.143} C_VEL
LIN {X 0,Y 516.51,Z 461.056,A -85,B 0,C 180,E1 -4945.315,E2 -4945.315} C_VEL
LIN {X 0,Y 516.515,Z 463.272,A -85,B 0,C 180,E1 -4946.097,E2 -4946.097} C_VEL
LIN {X 0,Y 516.475,Z 465.087,A -85,B 0,C 180,E1 -4946.878,E2 -4946.878} C_VEL
LIN {X 0,Y 516.425,Z 466.48,A -85,B 0,C 180,E1 -4947.658,E2 -4947.658} C_VEL
LIN {X 0,Y 516.361,Z 468.058,A -85,B 0,C 180,E1 -4949.218,E2 -4949.218} C_VEL
LIN {X 0,Y 516.354,Z 468.293,A -85,B 0,C 180,E1 -4949.998,E2 -4949.998} C_VEL
LIN {X 0,Y 516.347,Z 467.551,A -85,B 0,C 180,E1 -4951.558,E2 -4951.558} C_VEL
LIN {X 0,Y 516.503,Z 465.28,A -85,B 0,C 180,E1 -4953.118,E2 -4953.118} C_VEL
LIN {X 0,Y 516.55,Z 462.497,A -85,B 0,C 180,E1 -4954.29,E2 -4954.29} C_VEL
LIN {X 0,Y 516.593,Z 458.717,A -85,B 0,C 180,E1 -4955.463,E2 -4955.463} C_VEL
LIN {X 0,Y 516.711,Z 452.878,A -85,B 0,C 180,E1 -4956.827,E2 -4956.827} C_VEL
LIN {X 0,Y 516.947,Z 446.421,A -85,B 0,C 180,E1 -4958.008,E2 -4958.008} C_VEL
LIN {X 0,Y 517.207,Z 438.431,A -85,B 0,C 180,E1 -4959.185,E2 -4959.185} C_VEL
LIN {X 0,Y 517.448,Z 430.185,A -85,B 0,C 180,E1 -4960.168,E2 -4960.168} C_VEL
LIN {X 0,Y 517.741,Z 420.034,A -85,B 0,C 180,E1 -4961.151,E2 -4961.151} C_VEL
LIN {X 0,Y 518.036,Z 409.917,A -85,B 0,C 180,E1 -4961.942,E2 -4961.942} C_VEL
LIN {X 0,Y 518.247,Z 398.883,A -85,B 0,C 180,E1 -4962.629,E2 -4962.629} C_VEL
LIN {X 0,Y 518.51,Z 386.332,A -85,B 0,C 180,E1 -4963.22,E2 -4963.22} C_VEL
LIN {X 0,Y 518.648,Z 373.939,A -85,B 0,C 180,E1 -4963.64,E2 -4963.64} C_VEL
LIN {X 0,Y 517.385,Z 366.888,A -85,B 0,C 180,E1 -4963.847,E2 -4963.847} C_VEL
LIN {X 0,Y 516.786,Z 364.569,A -85,B 0,C 180,E1 -4963.916,E2 -4963.916} C_VEL
LIN {X 0,Y 516.756,Z 358.637,A -85,B 0,C 180,E1 -4966.593,E2 -4966.593} C_VEL
LIN {X 0,Y 516.799,Z 353.268,A -85,B 0,C 180,E1 -4969.047,E2 -4969.047} C_VEL
LIN {X 0,Y 516.879,Z 347.895,A -85,B 0,C 180,E1 -4971.536,E2 -4971.536} C_VEL
LIN {X 0,Y 516.993,Z 342.136,A -85,B 0,C 180,E1 -4974.383,E2 -4974.383} C_VEL
LIN {X 0,Y 517.084,Z 335.897,A -85,B 0,C 180,E1 -4977.521,E2 -4977.521} C_VEL
LIN {X 0,Y 517.209,Z 330.424,A -85,B 0,C 180,E1 -4980.18,E2 -4980.18} C_VEL
LIN {X 0,Y 517.284,Z 324.381,A -85,B 0,C 180,E1 -4982.916,E2 -4982.916} C_VEL
LIN {X 0,Y 517.203,Z 318.33,A -85,B 0,C 180,E1 -4985.382,E2 -4985.382} C_VEL
LIN {X 0,Y 516.957,Z 316.408,A -85,B 0,C 180,E1 -4986.131,E2 -4986.131} C_VEL
LIN {X 0,Y 516.875,Z 316.413,A -85,B 0,C 180,E1 -4989.191,E2 -4989.191} C_VEL
LIN {X 0,Y 516.891,Z 316.415,A -85,B 0,C 180,E1 -4991.774,E2 -4991.774} C_VEL
LIN {X 0,Y 516.908,Z 316.412,A -85,B 0,C 180,E1 -4995.008,E2 -4995.008} C_VEL
LIN {X 0,Y 516.913,Z 316.409,A -85,B 0,C 180,E1 -4998.395,E2 -4998.395} C_VEL
LIN {X 0,Y 516.892,Z 316.409,A -85,B 0,C 180,E1 -5001.285,E2 -5001.285} C_VEL
LIN {X 0,Y 516.87,Z 316.414,A -85,B 0,C 180,E1 -5004.219,E2 -5004.219} C_VEL
LIN {X 0,Y 516.874,Z 316.413,A -85,B 0,C 180,E1 -5007.051,E2 -5007.051} C_VEL
LIN {X 0,Y 516.871,Z 316.41,A -85,B 0,C 180,E1 -5009.795,E2 -5009.795} C_VEL
LIN {X 0,Y 516.91,Z 316.411,A -85,B 0,C 180,E1 -5012.466,E2 -5012.466} C_VEL
LIN {X 0,Y 516.908,Z 316.407,A -85,B 0,C 180,E1 -5015.071,E2 -5015.071} C_VEL
LIN {X 0,Y 516.89,Z 316.41,A -85,B 0,C 180,E1 -5017.622,E2 -5017.622} C_VEL
LIN {X 0,Y 516.909,Z 316.407,A -85,B 0,C 180,E1 -5020.129,E2 -5020.129} C_VEL
LIN {X 0,Y 516.904,Z 316.407,A -85,B 0,C 180,E1 -5022.595,E2 -5022.595} C_VEL
LIN {X 0,Y 516.917,Z 316.406,A -85,B 0,C 180,E1 -5025.029,E2 -5025.029} C_VEL
LIN {X 0,Y 516.979,Z 316.403,A -85,B 0,C 180,E1 -5028.234,E2 -5028.234} C_VEL
LIN {X 0,Y 516.952,Z 316.399,A -85,B 0,C 180,E1 -5031.399,E2 -5031.399} C_VEL
LIN {X 0,Y 517.021,Z 316.391,A -85,B 0,C 180,E1 -5034.54,E2 -5034.54} C_VEL
LIN {X 0,Y 517.051,Z 316.39,A -85,B 0,C 180,E1 -5037.663,E2 -5037.663} C_VEL
LIN {X 0,Y 517.073,Z 316.387,A -85,B 0,C 180,E1 -5040.778,E2 -5040.778} C_VEL
LIN {X 0,Y 517.025,Z 316.392,A -85,B 0,C 180,E1 -5043.117,E2 -5043.117} C_VEL
LIN {X 0,Y 516.994,Z 316.397,A -85,B 0,C 180,E1 -5046.243,E2 -5046.243} C_VEL
LIN {X 0,Y 516.938,Z 316.409,A -85,B 0,C 180,E1 -5049.389,E2 -5049.389} C_VEL
LIN {X 0,Y 516.957,Z 316.401,A -85,B 0,C 180,E1 -5051.824,E2 -5051.824} C_VEL
LIN {X 0,Y 516.92,Z 316.406,A -85,B 0,C 180,E1 -5055.148,E2 -5055.148} C_VEL
LIN {X 0,Y 516.906,Z 316.412,A -85,B 0,C 180,E1 -5058.223,E2 -5058.223} C_VEL
LIN {X 0,Y 516.893,Z 316.409,A -85,B 0,C 180,E1 -5060.702,E2 -5060.702} C_VEL
LIN {X 0,Y 516.88,Z 316.416,A -85,B 0,C 180,E1 -5063.223,E2 -5063.223} C_VEL
LIN {X 0,Y 516.915,Z 316.406,A -85,B 0,C 180,E1 -5066.197,E2 -5066.197} C_VEL
LIN {X 0,Y 516.898,Z 316.408,A -85,B 0,C 180,E1 -5069.306,E2 -5069.306} C_VEL
LIN {X 0,Y 516.882,Z 316.412,A -85,B 0,C 180,E1 -5072.546,E2 -5072.546} C_VEL
LIN {X 0,Y 516.864,Z 316.417,A -85,B 0,C 180,E1 -5075.334,E2 -5075.334} C_VEL
LIN {X 0,Y 516.865,Z 316.413,A -85,B 0,C 180,E1 -5077.945,E2 -5077.945} C_VEL
LIN {X 0,Y 516.863,Z 316.417,A -85,B 0,C 180,E1 -5080.743,E2 -5080.743} C_VEL
LIN {X 0,Y 516.862,Z 316.415,A -85,B 0,C 180,E1 -5082.833,E2 -5082.833} C_VEL
LIN {X 0,Y 516.904,Z 316.41,A -85,B 0,C 180,E1 -5085.012,E2 -5085.012} C_VEL
LIN {X 0,Y 516.912,Z 316.412,A -85,B 0,C 180,E1 -5088.399,E2 -5088.399} C_VEL
LIN {X 0,Y 516.938,Z 316.509,A -85,B 0,C 180,E1 -5089.919,E2 -5089.919} C_VEL
LIN {X 0,Y 521.003,Z 330.411,A -85,B 0,C 180,E1 -5092.737,E2 -5092.737} C_VEL
LIN {X 0,Y 523.09,Z 338.572,A -85,B 0,C 180,E1 -5094.255,E2 -5094.255} C_VEL
LIN {X 0,Y 522.296,Z 354.313,A -85,B 0,C 180,E1 -5096.694,E2 -5096.694} C_VEL
LIN {X 0,Y 521.274,Z 374.908,A -85,B 0,C 180,E1 -5099.778,E2 -5099.778} C_VEL
LIN {X 0,Y 520.447,Z 394.689,A -85,B 0,C 180,E1 -5102.672,E2 -5102.672} C_VEL
LIN {X 0,Y 519.614,Z 413.955,A -85,B 0,C 180,E1 -5105.426,E2 -5105.426} C_VEL
LIN {X 0,Y 519.399,Z 420.721,A -85,B 0,C 180,E1 -5106.385,E2 -5106.385} C_VEL
LIN {X 0,Y 522.848,Z 436.205,A -85,B 0,C 180,E1 -5106.792,E2 -5106.792} C_VEL
LIN {X 0,Y 522.636,Z 452.849,A -85,B 0,C 180,E1 -5107.133,E2 -5107.133} C_VEL
LIN {X 0,Y 522.202,Z 468.093,A -85,B 0,C 180,E1 -5107.588,E2 -5107.588} C_VEL
LIN {X 0,Y 521.707,Z 482.28,A -85,B 0,C 180,E1 -5108.141,E2 -5108.141} C_VEL
LIN {X 0,Y 521.149,Z 497.032,A -85,B 0,C 180,E1 -5108.857,E2 -5108.857} C_VEL
LIN {X 0,Y 520.52,Z 510.495,A -85,B 0,C 180,E1 -5109.657,E2 -5109.657} C_VEL
LIN {X 0,Y 519.791,Z 524.645,A -85,B 0,C 180,E1 -5110.657,E2 -5110.657} C_VEL
LIN {X 0,Y 519.16,Z 537.684,A -85,B 0,C 180,E1 -5111.748,E2 -5111.748} C_VEL
LIN {X 0,Y 518.446,Z 550.962,A -85,B 0,C 180,E1 -5113.057,E2 -5113.057} C_VEL
LIN {X 0,Y 517.896,Z 563.006,A -85,B 0,C 180,E1 -5114.469,E2 -5114.469} C_VEL
LIN {X 0,Y 517.396,Z 573.071,A -85,B 0,C 180,E1 -5115.85,E2 -5115.85} C_VEL
LIN {X 0,Y 517.026,Z 582.951,A -85,B 0,C 180,E1 -5117.441,E2 -5117.441} C_VEL
LIN {X 0,Y 516.729,Z 591.249,A -85,B 0,C 180,E1 -5119.025,E2 -5119.025} C_VEL
LIN {X 0,Y 516.489,Z 598.109,A -85,B 0,C 180,E1 -5120.604,E2 -5120.604} C_VEL
LIN {X 0,Y 516.408,Z 603.725,A -85,B 0,C 180,E1 -5122.18,E2 -5122.18} C_VEL
LIN {X 0,Y 516.321,Z 608.25,A -85,B 0,C 180,E1 -5123.751,E2 -5123.751} C_VEL
LIN {X 0,Y 516.225,Z 611.638,A -85,B 0,C 180,E1 -5125.317,E2 -5125.317} C_VEL
LIN {X 0,Y 516.267,Z 614.091,A -85,B 0,C 180,E1 -5126.881,E2 -5126.881} C_VEL
LIN {X 0,Y 516.186,Z 615.48,A -85,B 0,C 180,E1 -5128.442,E2 -5128.442} C_VEL
LIN {X 0,Y 516.149,Z 616,A -85,B 0,C 180,E1 -5130.002,E2 -5130.002} C_VEL
LIN {X 0,Y 516.186,Z 615.478,A -85,B 0,C 180,E1 -5131.562,E2 -5131.562} C_VEL
LIN {X 0,Y 516.267,Z 614.086,A -85,B 0,C 180,E1 -5133.123,E2 -5133.123} C_VEL
LIN {X 0,Y 516.226,Z 611.632,A -85,B 0,C 180,E1 -5134.687,E2 -5134.687} C_VEL
LIN {X 0,Y 516.37,Z 607.552,A -85,B 0,C 180,E1 -5136.509,E2 -5136.509} C_VEL
LIN {X 0,Y 516.42,Z 602.462,A -85,B 0,C 180,E1 -5138.217,E2 -5138.217} C_VEL
LIN {X 0,Y 516.622,Z 594.849,A -85,B 0,C 180,E1 -5140.188,E2 -5140.188} C_VEL
LIN {X 0,Y 516.917,Z 587.154,A -85,B 0,C 180,E1 -5141.789,E2 -5141.789} C_VEL
LIN {X 0,Y 517.206,Z 578.201,A -85,B 0,C 180,E1 -5143.358,E2 -5143.358} C_VEL
LIN {X 0,Y 517.737,Z 567.41,A -85,B 0,C 180,E1 -5144.948,E2 -5144.948} C_VEL
LIN {X 0,Y 518.139,Z 557.992,A -85,B 0,C 180,E1 -5146.146,E2 -5146.146} C_VEL
LIN {X 0,Y 518.645,Z 547.053,A -85,B 0,C 180,E1 -5147.346,E2 -5147.346} C_VEL
LIN {X 0,Y 519.312,Z 533.527,A -85,B 0,C 180,E1 -5148.619,E2 -5148.619} C_VEL
LIN {X 0,Y 520.055,Z 519.247,A -85,B 0,C 180,E1 -5149.747,E2 -5149.747} C_VEL
LIN {X 0,Y 520.772,Z 504,A -85,B 0,C 180,E1 -5150.749,E2 -5150.749} C_VEL
LIN {X 0,Y 521.471,Z 488.53,A -85,B 0,C 180,E1 -5151.577,E2 -5151.577} C_VEL
LIN {X 0,Y 522.002,Z 473.948,A -85,B 0,C 180,E1 -5152.198,E2 -5152.198} C_VEL
LIN {X 0,Y 522.503,Z 456.999,A -85,B 0,C 180,E1 -5152.755,E2 -5152.755} C_VEL
LIN {X 0,Y 522.872,Z 440.836,A -85,B 0,C 180,E1 -5153.126,E2 -5153.126} C_VEL
LIN {X 0,Y 522.681,Z 435.555,A -85,B 0,C 180,E1 -5153.227,E2 -5153.227} C_VEL
LIN {X 0,Y 519.395,Z 420.765,A -85,B 0,C 180,E1 -5153.609,E2 -5153.609} C_VEL
LIN {X 0,Y 520.121,Z 402.07,A -85,B 0,C 180,E1 -5156.267,E2 -5156.267} C_VEL
LIN {X 0,Y 520.997,Z 381.322,A -85,B 0,C 180,E1 -5159.276,E2 -5159.276} C_VEL
LIN {X 0,Y 522.079,Z 359.092,A -85,B 0,C 180,E1 -5162.58,E2 -5162.58} C_VEL
LIN {X 0,Y 523.146,Z 340.137,A -85,B 0,C 180,E1 -5165.517,E2 -5165.517} C_VEL
LIN {X 0,Y 522.941,Z 337.456,A -85,B 0,C 180,E1 -5165.987,E2 -5165.987} C_VEL
LIN {X 0,Y 520.436,Z 327.627,A -85,B 0,C 180,E1 -5168.137,E2 -5168.137} C_VEL
LIN {X 0,Y 518.449,Z 321.426,A -85,B 0,C 180,E1 -5169.81,E2 -5169.81} C_VEL
LIN {X 0,Y 516.909,Z 316.412,A -85,B 0,C 180,E1 -5171.535,E2 -5171.535} C_VEL
LIN {X 0,Y 516.9,Z 316.414,A -85,B 0,C 180,E1 -5175.008,E2 -5175.008} C_VEL
LIN {X 0,Y 516.906,Z 316.413,A -85,B 0,C 180,E1 -5178.401,E2 -5178.401} C_VEL
LIN {X 0,Y 516.881,Z 316.416,A -85,B 0,C 180,E1 -5181.284,E2 -5181.284} C_VEL
LIN {X 0,Y 516.919,Z 316.605,A -85,B 0,C 180,E1 -5182.402,E2 -5182.402} C_VEL
LIN {X 0,Y 517.802,Z 321.004,A -85,B 0,C 180,E1 -5184.526,E2 -5184.526} C_VEL
LIN {X 0,Y 517.9,Z 324.72,A -85,B 0,C 180,E1 -5186.195,E2 -5186.195} C_VEL
LIN {X 0,Y 517.708,Z 330.74,A -85,B 0,C 180,E1 -5188.945,E2 -5188.945} C_VEL
LIN {X 0,Y 517.555,Z 337.046,A -85,B 0,C 180,E1 -5191.965,E2 -5191.965} C_VEL
LIN {X 0,Y 517.371,Z 343.262,A -85,B 0,C 180,E1 -5195.096,E2 -5195.096} C_VEL
LIN {X 0,Y 517.252,Z 348.161,A -85,B 0,C 180,E1 -5197.639,E2 -5197.639} C_VEL
LIN {X 0,Y 517.085,Z 352.994,A -85,B 0,C 180,E1 -5200.136,E2 -5200.136} C_VEL
LIN {X 0,Y 516.922,Z 357.72,A -85,B 0,C 180,E1 -5202.596,E2 -5202.596} C_VEL
LIN {X 0,Y 516.885,Z 362.416,A -85,B 0,C 180,E1 -5205.029,E2 -5205.029} C_VEL
LIN {X 0,Y 516.826,Z 364.311,A -85,B 0,C 180,E1 -5205.951,E2 -5205.951} C_VEL
LIN {X 0,Y 518.665,Z 370.886,A -85,B 0,C 180,E1 -5206.183,E2 -5206.183} C_VEL
LIN {X 0,Y 519.107,Z 375.701,A -85,B 0,C 180,E1 -5206.345,E2 -5206.345} C_VEL
LIN {X 0,Y 518.828,Z 388.687,A -85,B 0,C 180,E1 -5206.836,E2 -5206.836} C_VEL
LIN {X 0,Y 518.408,Z 401.07,A -85,B 0,C 180,E1 -5207.473,E2 -5207.473} C_VEL
LIN {X 0,Y 518.127,Z 412.873,A -85,B 0,C 180,E1 -5208.261,E2 -5208.261} C_VEL
LIN {X 0,Y 517.776,Z 423.394,A -85,B 0,C 180,E1 -5209.145,E2 -5209.145} C_VEL
LIN {X 0,Y 517.493,Z 433.72,A -85,B 0,C 180,E1 -5210.226,E2 -5210.226} C_VEL
LIN {X 0,Y 517.217,Z 441.371,A -85,B 0,C 180,E1 -5211.207,E2 -5211.207} C_VEL
LIN {X 0,Y 516.994,Z 448.852,A -85,B 0,C 180,E1 -5212.384,E2 -5212.384} C_VEL
LIN {X 0,Y 516.774,Z 455.711,A -85,B 0,C 180,E1 -5213.754,E2 -5213.754} C_VEL
LIN {X 0,Y 516.595,Z 460.274,A -85,B 0,C 180,E1 -5214.927,E2 -5214.927} C_VEL
LIN {X 0,Y 516.619,Z 463.731,A -85,B 0,C 180,E1 -5216.1,E2 -5216.1} C_VEL
LIN {X 0,Y 516.536,Z 465.516,A -85,B 0,C 180,E1 -5216.88,E2 -5216.88} C_VEL
LIN {X 0,Y 516.479,Z 466.865,A -85,B 0,C 180,E1 -5217.661,E2 -5217.661} C_VEL
LIN {X 0,Y 516.363,Z 468.39,A -85,B 0,C 180,E1 -5219.22,E2 -5219.22} C_VEL
LIN {X 0,Y 516.362,Z 468.343,A -85,B 0,C 180,E1 -5220.78,E2 -5220.78} C_VEL
LIN {X 0,Y 516.425,Z 466.754,A -85,B 0,C 180,E1 -5222.34,E2 -5222.34} C_VEL
LIN {X 0,Y 516.478,Z 465.345,A -85,B 0,C 180,E1 -5223.12,E2 -5223.12} C_VEL
LIN {X 0,Y 516.52,Z 462.462,A -85,B 0,C 180,E1 -5224.292,E2 -5224.292} C_VEL
LIN {X 0,Y 516.552,Z 458.571,A -85,B 0,C 180,E1 -5225.465,E2 -5225.465} C_VEL
LIN {X 0,Y 516.716,Z 452.601,A -85,B 0,C 180,E1 -5226.83,E2 -5226.83} C_VEL
LIN {X 0,Y 516.908,Z 446.01,A -85,B 0,C 180,E1 -5228.011,E2 -5228.011} C_VEL
LIN {X 0,Y 517.111,Z 437.846,A -85,B 0,C 180,E1 -5229.189,E2 -5229.189} C_VEL
LIN {X 0,Y 517.321,Z 429.482,A -85,B 0,C 180,E1 -5230.173,E2 -5230.173} C_VEL
LIN {X 0,Y 517.646,Z 419.206,A -85,B 0,C 180,E1 -5231.156,E2 -5231.156} C_VEL
LIN {X 0,Y 517.953,Z 407.701,A -85,B 0,C 180,E1 -5232.037,E2 -5232.037} C_VEL
LIN {X 0,Y 518.266,Z 396.245,A -85,B 0,C 180,E1 -5232.73,E2 -5232.73} C_VEL
LIN {X 0,Y 518.521,Z 383.336,A -85,B 0,C 180,E1 -5233.322,E2 -5233.322} C_VEL
LIN {X 0,Y 518.528,Z 372.37,A -85,B 0,C 180,E1 -5233.696,E2 -5233.696} C_VEL
LIN {X 0,Y 516.459,Z 362.146,A -85,B 0,C 180,E1 -5234.028,E2 -5234.028} C_VEL
LIN {X 0,Y 516.501,Z 356.76,A -85,B 0,C 180,E1 -5236.604,E2 -5236.604} C_VEL
LIN {X 0,Y 516.626,Z 349.943,A -85,B 0,C 180,E1 -5239.883,E2 -5239.883} C_VEL
LIN {X 0,Y 516.739,Z 344.768,A -85,B 0,C 180,E1 -5242.385,E2 -5242.385} C_VEL
LIN {X 0,Y 516.783,Z 339.529,A -85,B 0,C 180,E1 -5244.935,E2 -5244.935} C_VEL
LIN {X 0,Y 516.912,Z 333.484,A -85,B 0,C 180,E1 -5247.901,E2 -5247.901} C_VEL
LIN {X 0,Y 516.978,Z 328.841,A -85,B 0,C 180,E1 -5250.199,E2 -5250.199} C_VEL
LIN {X 0,Y 517.094,Z 323.314,A -85,B 0,C 180,E1 -5252.933,E2 -5252.933} C_VEL
LIN {X 0,Y 517.031,Z 317.661,A -85,B 0,C 180,E1 -5255.768,E2 -5255.768} C_VEL
LIN {X 0,Y 516.937,Z 316.41,A -85,B 0,C 180,E1 -5256.436,E2 -5256.436} C_VEL
LIN {X 0,Y 516.879,Z 316.416,A -85,B 0,C 180,E1 -5259.722,E2 -5259.722} C_VEL
LIN {X 0,Y 516.915,Z 316.41,A -85,B 0,C 180,E1 -5261.775,E2 -5261.775} C_VEL
LIN {X 0,Y 516.883,Z 316.412,A -85,B 0,C 180,E1 -5264.728,E2 -5264.728} C_VEL
LIN {X 0,Y 516.25,Z 316.495,A -85,B 0,C 180,E1 -5265.379,E2 -5265.379} C_VEL
LIN {X 0,Y 513.409,Z 316.85,A -85,B 0,C 180,E1 -5266.435,E2 -5266.435} C_VEL
LIN {X 0,Y 510.986,Z 317.151,A -85,B 0,C 180,E1 -5267.285,E2 -5267.285} C_VEL
LIN {X 0,Y 509.941,Z 317.28,A -85,B 0,C 180,E1 -5267.942,E2 -5267.942} C_VEL
LIN {X 0,Y 509.856,Z 317.289,A -85,B 0,C 180,E1 -5268.165,E2 -5268.165} C_VEL
LIN {X 0,Y 509.846,Z 317.292,A -85,B 0,C 180,E1 -5270.646,E2 -5270.646} C_VEL
LIN {X 0,Y 509.88,Z 317.299,A -85,B 0,C 180,E1 -5273.85,E2 -5273.85} C_VEL
LIN {X 0,Y 510.306,Z 322.049,A -85,B 0,C 180,E1 -5275.724,E2 -5275.724} C_VEL
LIN {X 0,Y 510.206,Z 328.819,A -85,B 0,C 180,E1 -5278.654,E2 -5278.654} C_VEL
LIN {X 0,Y 510.106,Z 334.16,A -85,B 0,C 180,E1 -5281.168,E2 -5281.168} C_VEL
LIN {X 0,Y 510.039,Z 339.533,A -85,B 0,C 180,E1 -5283.835,E2 -5283.835} C_VEL
LIN {X 0,Y 509.937,Z 344.711,A -85,B 0,C 180,E1 -5286.44,E2 -5286.44} C_VEL
LIN {X 0,Y 509.84,Z 351.161,A -85,B 0,C 180,E1 -5289.614,E2 -5289.614} C_VEL
LIN {X 0,Y 509.79,Z 357.117,A -85,B 0,C 180,E1 -5292.343,E2 -5292.343} C_VEL
LIN {X 0,Y 509.764,Z 364.578,A -85,B 0,C 180,E1 -5295.63,E2 -5295.63} C_VEL
LIN {X 0,Y 509.827,Z 365.572,A -85,B 0,C 180,E1 -5295.987,E2 -5295.987} C_VEL
LIN {X 0,Y 511.777,Z 373.757,A -85,B 0,C 180,E1 -5296.232,E2 -5296.232} C_VEL
LIN {X 0,Y 511.671,Z 386.315,A -85,B 0,C 180,E1 -5296.647,E2 -5296.647} C_VEL
LIN {X 0,Y 511.419,Z 398.176,A -85,B 0,C 180,E1 -5297.196,E2 -5297.196} C_VEL
LIN {X 0,Y 511.201,Z 409.506,A -85,B 0,C 180,E1 -5297.884,E2 -5297.884} C_VEL
LIN {X 0,Y 510.907,Z 420.036,A -85,B 0,C 180,E1 -5298.694,E2 -5298.694} C_VEL
LIN {X 0,Y 510.529,Z 430.367,A -85,B 0,C 180,E1 -5299.689,E2 -5299.689} C_VEL
LIN {X 0,Y 510.3,Z 438.765,A -85,B 0,C 180,E1 -5300.685,E2 -5300.685} C_VEL
LIN {X 0,Y 510.015,Z 446.942,A -85,B 0,C 180,E1 -5301.878,E2 -5301.878} C_VEL
LIN {X 0,Y 509.798,Z 453.217,A -85,B 0,C 180,E1 -5303.019,E2 -5303.019} C_VEL
LIN {X 0,Y 509.63,Z 459.431,A -85,B 0,C 180,E1 -5304.459,E2 -5304.459} C_VEL
LIN {X 0,Y 509.527,Z 463.307,A -85,B 0,C 180,E1 -5305.647,E2 -5305.647} C_VEL
LIN {X 0,Y 509.468,Z 466.164,A -85,B 0,C 180,E1 -5306.835,E2 -5306.835} C_VEL
LIN {X 0,Y 509.428,Z 467.555,A -85,B 0,C 180,E1 -5307.626,E2 -5307.626} C_VEL
LIN {X 0,Y 509.364,Z 469.133,A -85,B 0,C 180,E1 -5309.208,E2 -5309.208} C_VEL
LIN {X 0,Y 509.355,Z 469.367,A -85,B 0,C 180,E1 -5309.998,E2 -5309.998} C_VEL
LIN {X 0,Y 509.364,Z 469.187,A -85,B 0,C 180,E1 -5310.789,E2 -5310.789} C_VEL
LIN {X 0,Y 509.43,Z 467.68,A -85,B 0,C 180,E1 -5312.37,E2 -5312.37} C_VEL
LIN {X 0,Y 509.507,Z 466.353,A -85,B 0,C 180,E1 -5313.161,E2 -5313.161} C_VEL
LIN {X 0,Y 509.559,Z 463.569,A -85,B 0,C 180,E1 -5314.348,E2 -5314.348} C_VEL
LIN {X 0,Y 509.623,Z 459.786,A -85,B 0,C 180,E1 -5315.538,E2 -5315.538} C_VEL
LIN {X 0,Y 509.742,Z 453.907,A -85,B 0,C 180,E1 -5316.929,E2 -5316.929} C_VEL
LIN {X 0,Y 510.007,Z 447.486,A -85,B 0,C 180,E1 -5318.118,E2 -5318.118} C_VEL
LIN {X 0,Y 510.291,Z 439.492,A -85,B 0,C 180,E1 -5319.311,E2 -5319.311} C_VEL
LIN {X 0,Y 510.549,Z 431.242,A -85,B 0,C 180,E1 -5320.307,E2 -5320.307} C_VEL
LIN {X 0,Y 510.859,Z 421.088,A -85,B 0,C 180,E1 -5321.303,E2 -5321.303} C_VEL
LIN {X 0,Y 511.175,Z 410.939,A -85,B 0,C 180,E1 -5322.107,E2 -5322.107} C_VEL
LIN {X 0,Y 511.391,Z 399.921,A -85,B 0,C 180,E1 -5322.801,E2 -5322.801} C_VEL
LIN {X 0,Y 511.654,Z 387.356,A -85,B 0,C 180,E1 -5323.4,E2 -5323.4} C_VEL
LIN {X 0,Y 511.813,Z 374.932,A -85,B 0,C 180,E1 -5323.826,E2 -5323.826} C_VEL
LIN {X 0,Y 510.735,Z 368.84,A -85,B 0,C 180,E1 -5324.011,E2 -5324.011} C_VEL
LIN {X 0,Y 509.805,Z 365.39,A -85,B 0,C 180,E1 -5324.128,E2 -5324.128} C_VEL
LIN {X 0,Y 509.744,Z 359.221,A -85,B 0,C 180,E1 -5326.828,E2 -5326.828} C_VEL
LIN {X 0,Y 509.79,Z 353.67,A -85,B 0,C 180,E1 -5329.319,E2 -5329.319} C_VEL
LIN {X 0,Y 509.855,Z 348.327,A -85,B 0,C 180,E1 -5331.847,E2 -5331.847} C_VEL
LIN {X 0,Y 509.979,Z 342.93,A -85,B 0,C 180,E1 -5334.557,E2 -5334.557} C_VEL
LIN {X 0,Y 510.057,Z 337.989,A -85,B 0,C 180,E1 -5337.043,E2 -5337.043} C_VEL
LIN {X 0,Y 510.18,Z 332.384,A -85,B 0,C 180,E1 -5339.789,E2 -5339.789} C_VEL
LIN {X 0,Y 510.265,Z 325.699,A -85,B 0,C 180,E1 -5342.842,E2 -5342.842} C_VEL
LIN {X 0,Y 510.204,Z 319.622,A -85,B 0,C 180,E1 -5345.345,E2 -5345.345} C_VEL
LIN {X 0,Y 509.905,Z 317.287,A -85,B 0,C 180,E1 -5346.295,E2 -5346.295} C_VEL
LIN {X 0,Y 509.822,Z 317.293,A -85,B 0,C 180,E1 -5349.468,E2 -5349.468} C_VEL
LIN {X 0,Y 509.801,Z 317.293,A -85,B 0,C 180,E1 -5352.489,E2 -5352.489} C_VEL
LIN {X 0,Y 509.842,Z 317.292,A -85,B 0,C 180,E1 -5355.33,E2 -5355.33} C_VEL
LIN {X 0,Y 509.857,Z 317.29,A -85,B 0,C 180,E1 -5358.574,E2 -5358.574} C_VEL
LIN {X 0,Y 509.843,Z 317.288,A -85,B 0,C 180,E1 -5361.661,E2 -5361.661} C_VEL
LIN {X 0,Y 509.825,Z 317.289,A -85,B 0,C 180,E1 -5364.621,E2 -5364.621} C_VEL
LIN {X 0,Y 509.84,Z 317.292,A -85,B 0,C 180,E1 -5367.479,E2 -5367.479} C_VEL
LIN {X 0,Y 509.837,Z 317.286,A -85,B 0,C 180,E1 -5370.272,E2 -5370.272} C_VEL
LIN {X 0,Y 509.868,Z 317.284,A -85,B 0,C 180,E1 -5372.943,E2 -5372.943} C_VEL
LIN {X 0,Y 509.875,Z 317.284,A -85,B 0,C 180,E1 -5375.574,E2 -5375.574} C_VEL
LIN {X 0,Y 509.833,Z 317.292,A -85,B 0,C 180,E1 -5378.149,E2 -5378.149} C_VEL
LIN {X 0,Y 509.84,Z 317.286,A -85,B 0,C 180,E1 -5380.68,E2 -5380.68} C_VEL
LIN {X 0,Y 509.859,Z 317.291,A -85,B 0,C 180,E1 -5383.174,E2 -5383.174} C_VEL
LIN {X 0,Y 509.841,Z 317.282,A -85,B 0,C 180,E1 -5385.633,E2 -5385.633} C_VEL
LIN {X 0,Y 509.917,Z 317.278,A -85,B 0,C 180,E1 -5388.874,E2 -5388.874} C_VEL
LIN {X 0,Y 509.928,Z 317.28,A -85,B 0,C 180,E1 -5392.078,E2 -5392.078} C_VEL
LIN {X 0,Y 509.97,Z 317.269,A -85,B 0,C 180,E1 -5394.464,E2 -5394.464} C_VEL
LIN {X 0,Y 510.023,Z 317.265,A -85,B 0,C 180,E1 -5397.63,E2 -5397.63} C_VEL
LIN {X 0,Y 510.043,Z 317.263,A -85,B 0,C 180,E1 -5400.789,E2 -5400.789} C_VEL
LIN {X 0,Y 509.965,Z 317.271,A -85,B 0,C 180,E1 -5403.16,E2 -5403.16} C_VEL
LIN {X 0,Y 509.96,Z 317.273,A -85,B 0,C 180,E1 -5406.33,E2 -5406.33} C_VEL
LIN {X 0,Y 509.896,Z 317.281,A -85,B 0,C 180,E1 -5408.72,E2 -5408.72} C_VEL
LIN {X 0,Y 509.925,Z 317.277,A -85,B 0,C 180,E1 -5411.931,E2 -5411.931} C_VEL
LIN {X 0,Y 509.867,Z 317.284,A -85,B 0,C 180,E1 -5415.242,E2 -5415.242} C_VEL
LIN {X 0,Y 509.886,Z 317.288,A -85,B 0,C 180,E1 -5418.01,E2 -5418.01} C_VEL
LIN {X 0,Y 509.838,Z 317.288,A -85,B 0,C 180,E1 -5421.002,E2 -5421.002} C_VEL
LIN {X 0,Y 509.838,Z 317.291,A -85,B 0,C 180,E1 -5423.563,E2 -5423.563} C_VEL
LIN {X 0,Y 509.884,Z 317.283,A -85,B 0,C 180,E1 -5426.379,E2 -5426.379} C_VEL
LIN {X 0,Y 509.852,Z 317.289,A -85,B 0,C 180,E1 -5428.845,E2 -5428.845} C_VEL
LIN {X 0,Y 509.804,Z 317.294,A -85,B 0,C 180,E1 -5431.591,E2 -5431.591} C_VEL
LIN {X 0,Y 509.834,Z 317.29,A -85,B 0,C 180,E1 -5434.414,E2 -5434.414} C_VEL
LIN {X 0,Y 509.802,Z 317.297,A -85,B 0,C 180,E1 -5437.342,E2 -5437.342} C_VEL
LIN {X 0,Y 509.817,Z 317.292,A -85,B 0,C 180,E1 -5440.384,E2 -5440.384} C_VEL
LIN {X 0,Y 509.802,Z 317.292,A -85,B 0,C 180,E1 -5443.064,E2 -5443.064} C_VEL
LIN {X 0,Y 509.812,Z 317.297,A -85,B 0,C 180,E1 -5445.794,E2 -5445.794} C_VEL
LIN {X 0,Y 509.854,Z 317.291,A -85,B 0,C 180,E1 -5448.578,E2 -5448.578} C_VEL
LIN {X 0,Y 509.873,Z 317.371,A -85,B 0,C 180,E1 -5449.362,E2 -5449.362} C_VEL
LIN {X 0,Y 514.245,Z 332.121,A -85,B 0,C 180,E1 -5452.435,E2 -5452.435} C_VEL
LIN {X 0,Y 516.334,Z 340.107,A -85,B 0,C 180,E1 -5453.968,E2 -5453.968} C_VEL
LIN {X 0,Y 516.399,Z 343.655,A -85,B 0,C 180,E1 -5454.56,E2 -5454.56} C_VEL
LIN {X 0,Y 515.401,Z 360.69,A -85,B 0,C 180,E1 -5457.204,E2 -5457.204} C_VEL
LIN {X 0,Y 514.341,Z 381.351,A -85,B 0,C 180,E1 -5460.312,E2 -5460.312} C_VEL
LIN {X 0,Y 513.441,Z 400.617,A -85,B 0,C 180,E1 -5463.15,E2 -5463.15} C_VEL
LIN {X 0,Y 512.653,Z 420.834,A -85,B 0,C 180,E1 -5466.065,E2 -5466.065} C_VEL
LIN {X 0,Y 516.357,Z 438.36,A -85,B 0,C 180,E1 -5466.521,E2 -5466.521} C_VEL
LIN {X 0,Y 515.938,Z 456.147,A -85,B 0,C 180,E1 -5466.914,E2 -5466.914} C_VEL
LIN {X 0,Y 515.479,Z 471.79,A -85,B 0,C 180,E1 -5467.418,E2 -5467.418} C_VEL
LIN {X 0,Y 514.96,Z 485.959,A -85,B 0,C 180,E1 -5468.012,E2 -5468.012} C_VEL
LIN {X 0,Y 514.298,Z 500.558,A -85,B 0,C 180,E1 -5468.772,E2 -5468.772} C_VEL
LIN {X 0,Y 513.586,Z 515.033,A -85,B 0,C 180,E1 -5469.684,E2 -5469.684} C_VEL
LIN {X 0,Y 512.879,Z 528.494,A -85,B 0,C 180,E1 -5470.698,E2 -5470.698} C_VEL
LIN {X 0,Y 512.079,Z 542.065,A -85,B 0,C 180,E1 -5471.912,E2 -5471.912} C_VEL
LIN {X 0,Y 511.41,Z 554.523,A -85,B 0,C 180,E1 -5473.229,E2 -5473.229} C_VEL
LIN {X 0,Y 510.808,Z 566.158,A -85,B 0,C 180,E1 -5474.672,E2 -5474.672} C_VEL
LIN {X 0,Y 510.338,Z 575.753,A -85,B 0,C 180,E1 -5476.057,E2 -5476.057} C_VEL
LIN {X 0,Y 509.921,Z 585.177,A -85,B 0,C 180,E1 -5477.667,E2 -5477.667} C_VEL
LIN {X 0,Y 509.632,Z 593.062,A -85,B 0,C 180,E1 -5479.273,E2 -5479.273} C_VEL
LIN {X 0,Y 509.4,Z 599.635,A -85,B 0,C 180,E1 -5480.873,E2 -5480.873} C_VEL
LIN {X 0,Y 509.314,Z 604.961,A -85,B 0,C 180,E1 -5482.47,E2 -5482.47} C_VEL
LIN {X 0,Y 509.253,Z 608.25,A -85,B 0,C 180,E1 -5483.663,E2 -5483.663} C_VEL
LIN {X 0,Y 509.141,Z 611.638,A -85,B 0,C 180,E1 -5485.251,E2 -5485.251} C_VEL
LIN {X 0,Y 509.183,Z 614.092,A -85,B 0,C 180,E1 -5486.837,E2 -5486.837} C_VEL
LIN {X 0,Y 509.106,Z 615.48,A -85,B 0,C 180,E1 -5488.42,E2 -5488.42} C_VEL
LIN {X 0,Y 509.061,Z 616,A -85,B 0,C 180,E1 -5490.002,E2 -5490.002} C_VEL
LIN {X 0,Y 509.107,Z 615.478,A -85,B 0,C 180,E1 -5491.584,E2 -5491.584} C_VEL
LIN {X 0,Y 509.184,Z 614.086,A -85,B 0,C 180,E1 -5493.167,E2 -5493.167} C_VEL
LIN {X 0,Y 509.142,Z 611.632,A -85,B 0,C 180,E1 -5494.753,E2 -5494.753} C_VEL
LIN {X 0,Y 509.266,Z 607.876,A -85,B 0,C 180,E1 -5496.479,E2 -5496.479} C_VEL
LIN {X 0,Y 509.354,Z 602.462,A -85,B 0,C 180,E1 -5498.332,E2 -5498.332} C_VEL
LIN {X 0,Y 509.572,Z 594.849,A -85,B 0,C 180,E1 -5500.33,E2 -5500.33} C_VEL
LIN {X 0,Y 509.918,Z 586.244,A -85,B 0,C 180,E1 -5502.135,E2 -5502.135} C_VEL
LIN {X 0,Y 510.262,Z 576.966,A -85,B 0,C 180,E1 -5503.746,E2 -5503.746} C_VEL
LIN {X 0,Y 510.798,Z 566.215,A -85,B 0,C 180,E1 -5505.32,E2 -5505.32} C_VEL
LIN {X 0,Y 511.416,Z 554.491,A -85,B 0,C 180,E1 -5506.775,E2 -5506.775} C_VEL
LIN {X 0,Y 512.061,Z 542.027,A -85,B 0,C 180,E1 -5508.093,E2 -5508.093} C_VEL
LIN {X 0,Y 512.863,Z 528.448,A -85,B 0,C 180,E1 -5509.307,E2 -5509.307} C_VEL
LIN {X 0,Y 513.59,Z 514.974,A -85,B 0,C 180,E1 -5510.32,E2 -5510.32} C_VEL
LIN {X 0,Y 514.299,Z 500.486,A -85,B 0,C 180,E1 -5511.232,E2 -5511.232} C_VEL
LIN {X 0,Y 515.032,Z 484.745,A -85,B 0,C 180,E1 -5512.041,E2 -5512.041} C_VEL
LIN {X 0,Y 515.546,Z 470.543,A -85,B 0,C 180,E1 -5512.63,E2 -5512.63} C_VEL
LIN {X 0,Y 516.065,Z 454.463,A -85,B 0,C 180,E1 -5513.128,E2 -5513.128} C_VEL
LIN {X 0,Y 516.403,Z 438.129,A -85,B 0,C 180,E1 -5513.481,E2 -5513.481} C_VEL
LIN {X 0,Y 512.598,Z 420.724,A -85,B 0,C 180,E1 -5513.947,E2 -5513.947} C_VEL
LIN {X 0,Y 513.398,Z 402.07,A -85,B 0,C 180,E1 -5516.637,E2 -5516.637} C_VEL
LIN {X 0,Y 514.327,Z 381.322,A -85,B 0,C 180,E1 -5519.693,E2 -5519.693} C_VEL
LIN {X 0,Y 515.432,Z 360.501,A -85,B 0,C 180,E1 -5522.821,E2 -5522.821} C_VEL
LIN {X 0,Y 516.072,Z 350.378,A -85,B 0,C 180,E1 -5524.415,E2 -5524.415} C_VEL
LIN {X 0,Y 516.629,Z 341.764,A -85,B 0,C 180,E1 -5525.801,E2 -5525.801} C_VEL
LIN {X 0,Y 515.651,Z 336.723,A -85,B 0,C 180,E1 -5526.849,E2 -5526.849} C_VEL
LIN {X 0,Y 514.099,Z 330.797,A -85,B 0,C 180,E1 -5528.185,E2 -5528.185} C_VEL
LIN {X 0,Y 512.243,Z 324.913,A -85,B 0,C 180,E1 -5529.797,E2 -5529.797} C_VEL
LIN {X 0,Y 510.787,Z 320.362,A -85,B 0,C 180,E1 -5531.335,E2 -5531.335} C_VEL
LIN {X 0,Y 509.834,Z 317.294,A -85,B 0,C 180,E1 -5532.703,E2 -5532.703} C_VEL
LIN {X 0,Y 509.826,Z 317.294,A -85,B 0,C 180,E1 -5535.794,E2 -5535.794} C_VEL
LIN {X 0,Y 509.848,Z 317.292,A -85,B 0,C 180,E1 -5538.574,E2 -5538.574} C_VEL
LIN {X 0,Y 509.846,Z 317.419,A -85,B 0,C 180,E1 -5541.536,E2 -5541.536} C_VEL
LIN {X 0,Y 510.961,Z 322.489,A -85,B 0,C 180,E1 -5544.246,E2 -5544.246} C_VEL
LIN {X 0,Y 511.052,Z 326.501,A -85,B 0,C 180,E1 -5546.155,E2 -5546.155} C_VEL
LIN {X 0,Y 510.773,Z 333.387,A -85,B 0,C 180,E1 -5549.396,E2 -5549.396} C_VEL
LIN {X 0,Y 510.614,Z 338.897,A -85,B 0,C 180,E1 -5552.098,E2 -5552.098} C_VEL
LIN {X 0,Y 510.436,Z 345.213,A -85,B 0,C 180,E1 -5555.332,E2 -5555.332} C_VEL
LIN {X 0,Y 510.277,Z 350.655,A -85,B 0,C 180,E1 -5558.169,E2 -5558.169} C_VEL
LIN {X 0,Y 510.1,Z 355.467,A -85,B 0,C 180,E1 -5560.691,E2 -5560.691} C_VEL
LIN {X 0,Y 509.928,Z 360.22,A -85,B 0,C 180,E1 -5563.177,E2 -5563.177} C_VEL
LIN {X 0,Y 509.829,Z 365.029,A -85,B 0,C 180,E1 -5565.684,E2 -5565.684} C_VEL
LIN {X 0,Y 512.276,Z 373.81,A -85,B 0,C 180,E1 -5566.02,E2 -5566.02} C_VEL
LIN {X 0,Y 512.144,Z 387.14,A -85,B 0,C 180,E1 -5566.51,E2 -5566.51} C_VEL
LIN {X 0,Y 511.76,Z 399.626,A -85,B 0,C 180,E1 -5567.126,E2 -5567.126} C_VEL
LIN {X 0,Y 511.426,Z 410.754,A -85,B 0,C 180,E1 -5567.84,E2 -5567.84} C_VEL
LIN {X 0,Y 511.11,Z 421.495,A -85,B 0,C 180,E1 -5568.7,E2 -5568.7} C_VEL
LIN {X 0,Y 510.736,Z 431.584,A -85,B 0,C 180,E1 -5569.695,E2 -5569.695} C_VEL
LIN {X 0,Y 510.422,Z 441.233,A -85,B 0,C 180,E1 -5570.89,E2 -5570.89} C_VEL
LIN {X 0,Y 510.112,Z 448.998,A -85,B 0,C 180,E1 -5572.081,E2 -5572.081} C_VEL
LIN {X 0,Y 509.872,Z 455.43,A -85,B 0,C 180,E1 -5573.314,E2 -5573.314} C_VEL
LIN {X 0,Y 509.68,Z 460.169,A -85,B 0,C 180,E1 -5574.461,E2 -5574.461} C_VEL
LIN {X 0,Y 509.623,Z 463.966,A -85,B 0,C 180,E1 -5575.65,E2 -5575.65} C_VEL
LIN {X 0,Y 509.557,Z 466.756,A -85,B 0,C 180,E1 -5576.838,E2 -5576.838} C_VEL
LIN {X 0,Y 509.505,Z 468.094,A -85,B 0,C 180,E1 -5577.629,E2 -5577.629} C_VEL
LIN {X 0,Y 509.367,Z 469.588,A -85,B 0,C 180,E1 -5579.21,E2 -5579.21} C_VEL
LIN {X 0,Y 509.356,Z 469.746,A -85,B 0,C 180,E1 -5580,E2 -5580} C_VEL
LIN {X 0,Y 509.411,Z 468.885,A -85,B 0,C 180,E1 -5581.581,E2 -5581.581} C_VEL
LIN {X 0,Y 509.428,Z 467.872,A -85,B 0,C 180,E1 -5582.372,E2 -5582.372} C_VEL
LIN {X 0,Y 509.501,Z 466.439,A -85,B 0,C 180,E1 -5583.163,E2 -5583.163} C_VEL
LIN {X 0,Y 509.519,Z 463.52,A -85,B 0,C 180,E1 -5584.351,E2 -5584.351} C_VEL
LIN {X 0,Y 509.568,Z 459.584,A -85,B 0,C 180,E1 -5585.541,E2 -5585.541} C_VEL
LIN {X 0,Y 509.742,Z 453.554,A -85,B 0,C 180,E1 -5586.927,E2 -5586.927} C_VEL
LIN {X 0,Y 509.949,Z 446.938,A -85,B 0,C 180,E1 -5588.121,E2 -5588.121} C_VEL
LIN {X 0,Y 510.168,Z 438.714,A -85,B 0,C 180,E1 -5589.316,E2 -5589.316} C_VEL
LIN {X 0,Y 510.391,Z 430.315,A -85,B 0,C 180,E1 -5590.312,E2 -5590.312} C_VEL
LIN {X 0,Y 510.741,Z 420.014,A -85,B 0,C 180,E1 -5591.308,E2 -5591.308} C_VEL
LIN {X 0,Y 511.055,Z 408.617,A -85,B 0,C 180,E1 -5592.193,E2 -5592.193} C_VEL
LIN {X 0,Y 511.409,Z 397.05,A -85,B 0,C 180,E1 -5592.904,E2 -5592.904} C_VEL
LIN {X 0,Y 511.678,Z 384.237,A -85,B 0,C 180,E1 -5593.503,E2 -5593.503} C_VEL
LIN {X 0,Y 511.728,Z 373.458,A -85,B 0,C 180,E1 -5593.882,E2 -5593.882} C_VEL
LIN {X 0,Y 509.421,Z 362.508,A -85,B 0,C 180,E1 -5594.252,E2 -5594.252} C_VEL
LIN {X 0,Y 509.452,Z 357.137,A -85,B 0,C 180,E1 -5596.84,E2 -5596.84} C_VEL
LIN {X 0,Y 509.525,Z 351.964,A -85,B 0,C 180,E1 -5599.332,E2 -5599.332} C_VEL
LIN {X 0,Y 509.714,Z 345.404,A -85,B 0,C 180,E1 -5602.509,E2 -5602.509} C_VEL
LIN {X 0,Y 509.746,Z 339.727,A -85,B 0,C 180,E1 -5605.303,E2 -5605.303} C_VEL
LIN {X 0,Y 509.888,Z 334.08,A -85,B 0,C 180,E1 -5608.097,E2 -5608.097} C_VEL
LIN {X 0,Y 509.963,Z 328.942,A -85,B 0,C 180,E1 -5610.658,E2 -5610.658} C_VEL
LIN {X 0,Y 510.087,Z 323.362,A -85,B 0,C 180,E1 -5613.444,E2 -5613.444} C_VEL
LIN {X 0,Y 510.067,Z 319.051,A -85,B 0,C 180,E1 -5615.615,E2 -5615.615} C_VEL
LIN {X 0,Y 509.89,Z 317.287,A -85,B 0,C 180,E1 -5616.555,E2 -5616.555} C_VEL
LIN {X 0,Y 509.832,Z 317.293,A -85,B 0,C 180,E1 -5619.469,E2 -5619.469} C_VEL
LIN {X 0,Y 509.825,Z 317.294,A -85,B 0,C 180,E1 -5622.491,E2 -5622.491} C_VEL
LIN {X 0,Y 509.847,Z 317.292,A -85,B 0,C 180,E1 -5625.33,E2 -5625.33} C_VEL
LIN {X 0,Y 509.856,Z 317.289,A -85,B 0,C 180,E1 -5628.165,E2 -5628.165} C_VEL
LIN {X 0,Y 509.187,Z 317.374,A -85,B 0,C 180,E1 -5628.824,E2 -5628.824} C_VEL
LIN {X 0,Y 506.332,Z 317.729,A -85,B 0,C 180,E1 -5629.895,E2 -5629.895} C_VEL
LIN {X 0,Y 503.919,Z 318.032,A -85,B 0,C 180,E1 -5630.757,E2 -5630.757} C_VEL
LIN {X 0,Y 502.882,Z 318.161,A -85,B 0,C 180,E1 -5631.423,E2 -5631.423} C_VEL
LIN {X 0,Y 502.796,Z 318.17,A -85,B 0,C 180,E1 -5631.648,E2 -5631.648} C_VEL
LIN {X 0,Y 502.845,Z 318.24,A -85,B 0,C 180,E1 -5633.744,E2 -5633.744} C_VEL
LIN {X 0,Y 503.284,Z 322.624,A -85,B 0,C 180,E1 -5635.477,E2 -5635.477} C_VEL
LIN {X 0,Y 503.23,Z 328.395,A -85,B 0,C 180,E1 -5637.946,E2 -5637.946} C_VEL
LIN {X 0,Y 503.116,Z 334.39,A -85,B 0,C 180,E1 -5640.729,E2 -5640.729} C_VEL
LIN {X 0,Y 503.031,Z 339.888,A -85,B 0,C 180,E1 -5643.442,E2 -5643.442} C_VEL
LIN {X 0,Y 502.941,Z 345.164,A -85,B 0,C 180,E1 -5646.092,E2 -5646.092} C_VEL
LIN {X 0,Y 502.836,Z 352.162,A -85,B 0,C 180,E1 -5649.547,E2 -5649.547} C_VEL
LIN {X 0,Y 502.795,Z 357.644,A -85,B 0,C 180,E1 -5652.089,E2 -5652.089} C_VEL
LIN {X 0,Y 502.768,Z 365.358,A -85,B 0,C 180,E1 -5655.425,E2 -5655.425} C_VEL
LIN {X 0,Y 502.806,Z 366.199,A -85,B 0,C 180,E1 -5655.775,E2 -5655.775} C_VEL
LIN {X 0,Y 504.975,Z 374.991,A -85,B 0,C 180,E1 -5656.048,E2 -5656.048} C_VEL
LIN {X 0,Y 504.83,Z 387.372,A -85,B 0,C 180,E1 -5656.462,E2 -5656.462} C_VEL
LIN {X 0,Y 504.57,Z 399.24,A -85,B 0,C 180,E1 -5657.019,E2 -5657.019} C_VEL
LIN {X 0,Y 504.343,Z 410.549,A -85,B 0,C 180,E1 -5657.715,E2 -5657.715} C_VEL
LIN {X 0,Y 504.03,Z 421.105,A -85,B 0,C 180,E1 -5658.538,E2 -5658.538} C_VEL
LIN {X 0,Y 503.653,Z 431.435,A -85,B 0,C 180,E1 -5659.547,E2 -5659.547} C_VEL
LIN {X 0,Y 503.383,Z 439.837,A -85,B 0,C 180,E1 -5660.556,E2 -5660.556} C_VEL
LIN {X 0,Y 503.07,Z 448.016,A -85,B 0,C 180,E1 -5661.765,E2 -5661.765} C_VEL
LIN {X 0,Y 502.837,Z 454.232,A -85,B 0,C 180,E1 -5662.909,E2 -5662.909} C_VEL
LIN {X 0,Y 502.741,Z 458.963,A -85,B 0,C 180,E1 -5663.98,E2 -5663.98} C_VEL
LIN {X 0,Y 502.519,Z 463.21,A -85,B 0,C 180,E1 -5665.185,E2 -5665.185} C_VEL
LIN {X 0,Y 502.511,Z 465.426,A -85,B 0,C 180,E1 -5665.988,E2 -5665.988} C_VEL
LIN {X 0,Y 502.461,Z 467.241,A -85,B 0,C 180,E1 -5666.791,E2 -5666.791} C_VEL
LIN {X 0,Y 502.429,Z 468.63,A -85,B 0,C 180,E1 -5667.593,E2 -5667.593} C_VEL
LIN {X 0,Y 502.365,Z 470.207,A -85,B 0,C 180,E1 -5669.196,E2 -5669.196} C_VEL
LIN {X 0,Y 502.353,Z 470.441,A -85,B 0,C 180,E1 -5669.998,E2 -5669.998} C_VEL
LIN {X 0,Y 502.364,Z 470.261,A -85,B 0,C 180,E1 -5670.8,E2 -5670.8} C_VEL
LIN {X 0,Y 502.431,Z 468.753,A -85,B 0,C 180,E1 -5672.403,E2 -5672.403} C_VEL
LIN {X 0,Y 502.525,Z 467.423,A -85,B 0,C 180,E1 -5673.205,E2 -5673.205} C_VEL
LIN {X 0,Y 502.582,Z 464.64,A -85,B 0,C 180,E1 -5674.409,E2 -5674.409} C_VEL
LIN {X 0,Y 502.651,Z 460.856,A -85,B 0,C 180,E1 -5675.615,E2 -5675.615} C_VEL
LIN {X 0,Y 502.778,Z 454.923,A -85,B 0,C 180,E1 -5677.037,E2 -5677.037} C_VEL
LIN {X 0,Y 503.063,Z 448.553,A -85,B 0,C 180,E1 -5678.231,E2 -5678.231} C_VEL
LIN {X 0,Y 503.377,Z 440.554,A -85,B 0,C 180,E1 -5679.44,E2 -5679.44} C_VEL
LIN {X 0,Y 503.653,Z 432.301,A -85,B 0,C 180,E1 -5680.449,E2 -5680.449} C_VEL
LIN {X 0,Y 503.978,Z 422.144,A -85,B 0,C 180,E1 -5681.46,E2 -5681.46} C_VEL
LIN {X 0,Y 504.314,Z 411.983,A -85,B 0,C 180,E1 -5682.275,E2 -5682.275} C_VEL
LIN {X 0,Y 504.541,Z 400.962,A -85,B 0,C 180,E1 -5682.978,E2 -5682.978} C_VEL
LIN {X 0,Y 504.798,Z 388.386,A -85,B 0,C 180,E1 -5683.586,E2 -5683.586} C_VEL
LIN {X 0,Y 504.993,Z 375.927,A -85,B 0,C 180,E1 -5684.017,E2 -5684.017} C_VEL
LIN {X 0,Y 503.906,Z 370.193,A -85,B 0,C 180,E1 -5684.196,E2 -5684.196} C_VEL
LIN {X 0,Y 502.795,Z 366.22,A -85,B 0,C 180,E1 -5684.329,E2 -5684.329} C_VEL
LIN {X 0,Y 502.723,Z 359.766,A -85,B 0,C 180,E1 -5687.07,E2 -5687.07} C_VEL
LIN {X 0,Y 502.789,Z 354.188,A -85,B 0,C 180,E1 -5689.599,E2 -5689.599} C_VEL
LIN {X 0,Y 502.877,Z 347.726,A -85,B 0,C 180,E1 -5692.721,E2 -5692.721} C_VEL
LIN {X 0,Y 503.009,Z 341.87,A -85,B 0,C 180,E1 -5695.664,E2 -5695.664} C_VEL
LIN {X 0,Y 503.08,Z 336.484,A -85,B 0,C 180,E1 -5698.355,E2 -5698.355} C_VEL
LIN {X 0,Y 503.211,Z 330.715,A -85,B 0,C 180,E1 -5701.112,E2 -5701.112} C_VEL
LIN {X 0,Y 503.297,Z 324.252,A -85,B 0,C 180,E1 -5703.953,E2 -5703.953} C_VEL
LIN {X 0,Y 503.099,Z 319.358,A -85,B 0,C 180,E1 -5705.921,E2 -5705.921} C_VEL
LIN {X 0,Y 502.839,Z 318.167,A -85,B 0,C 180,E1 -5706.438,E2 -5706.438} C_VEL
LIN {X 0,Y 502.776,Z 318.173,A -85,B 0,C 180,E1 -5709.752,E2 -5709.752} C_VEL
LIN {X 0,Y 502.789,Z 318.168,A -85,B 0,C 180,E1 -5712.197,E2 -5712.197} C_VEL
LIN {X 0,Y 502.786,Z 318.169,A -85,B 0,C 180,E1 -5715.466,E2 -5715.466} C_VEL
LIN {X 0,Y 502.822,Z 318.161,A -85,B 0,C 180,E1 -5717.863,E2 -5717.863} C_VEL
LIN {X 0,Y 502.81,Z 318.164,A -85,B 0,C 180,E1 -5721.024,E2 -5721.024} C_VEL
LIN {X 0,Y 502.765,Z 318.172,A -85,B 0,C 180,E1 -5724.166,E2 -5724.166} C_VEL
LIN {X 0,Y 502.812,Z 318.164,A -85,B 0,C 180,E1 -5726.991,E2 -5726.991} C_VEL
LIN {X 0,Y 502.794,Z 318.163,A -85,B 0,C 180,E1 -5730.063,E2 -5730.063} C_VEL
LIN {X 0,Y 502.815,Z 318.168,A -85,B 0,C 180,E1 -5732.532,E2 -5732.532} C_VEL
LIN {X 0,Y 502.819,Z 318.162,A -85,B 0,C 180,E1 -5735.294,E2 -5735.294} C_VEL
LIN {X 0,Y 502.799,Z 318.166,A -85,B 0,C 180,E1 -5737.827,E2 -5737.827} C_VEL
LIN {X 0,Y 502.801,Z 318.162,A -85,B 0,C 180,E1 -5740.399,E2 -5740.399} C_VEL
LIN {X 0,Y 502.809,Z 318.166,A -85,B 0,C 180,E1 -5742.93,E2 -5742.93} C_VEL
LIN {X 0,Y 502.821,Z 318.157,A -85,B 0,C 180,E1 -5745.428,E2 -5745.428} C_VEL
LIN {X 0,Y 502.886,Z 318.155,A -85,B 0,C 180,E1 -5748.717,E2 -5748.717} C_VEL
LIN {X 0,Y 502.882,Z 318.159,A -85,B 0,C 180,E1 -5751.966,E2 -5751.966} C_VEL
LIN {X 0,Y 502.924,Z 318.147,A -85,B 0,C 180,E1 -5754.386,E2 -5754.386} C_VEL
LIN {X 0,Y 502.994,Z 318.141,A -85,B 0,C 180,E1 -5757.597,E2 -5757.597} C_VEL
LIN {X 0,Y 502.997,Z 318.138,A -85,B 0,C 180,E1 -5760,E2 -5760} C_VEL
LIN {X 0,Y 503.005,Z 318.143,A -85,B 0,C 180,E1 -5762.402,E2 -5762.402} C_VEL
LIN {X 0,Y 502.942,Z 318.15,A -85,B 0,C 180,E1 -5765.613,E2 -5765.613} C_VEL
LIN {X 0,Y 502.877,Z 318.156,A -85,B 0,C 180,E1 -5768.033,E2 -5768.033} C_VEL
LIN {X 0,Y 502.877,Z 318.16,A -85,B 0,C 180,E1 -5771.283,E2 -5771.283} C_VEL
LIN {X 0,Y 502.823,Z 318.167,A -85,B 0,C 180,E1 -5774.571,E2 -5774.571} C_VEL
LIN {X 0,Y 502.855,Z 318.162,A -85,B 0,C 180,E1 -5777.907,E2 -5777.907} C_VEL
LIN {X 0,Y 502.807,Z 318.164,A -85,B 0,C 180,E1 -5780.538,E2 -5780.538} C_VEL
LIN {X 0,Y 502.796,Z 318.168,A -85,B 0,C 180,E1 -5783.04,E2 -5783.04} C_VEL
LIN {X 0,Y 502.816,Z 318.163,A -85,B 0,C 180,E1 -5785.677,E2 -5785.677} C_VEL
LIN {X 0,Y 502.815,Z 318.166,A -85,B 0,C 180,E1 -5788.374,E2 -5788.374} C_VEL
LIN {X 0,Y 502.774,Z 318.169,A -85,B 0,C 180,E1 -5791.501,E2 -5791.501} C_VEL
LIN {X 0,Y 502.786,Z 318.167,A -85,B 0,C 180,E1 -5794.446,E2 -5794.446} C_VEL
LIN {X 0,Y 502.763,Z 318.173,A -85,B 0,C 180,E1 -5797.18,E2 -5797.18} C_VEL
LIN {X 0,Y 502.768,Z 318.169,A -85,B 0,C 180,E1 -5800.017,E2 -5800.017} C_VEL
LIN {X 0,Y 502.783,Z 318.167,A -85,B 0,C 180,E1 -5802.201,E2 -5802.201} C_VEL
LIN {X 0,Y 502.782,Z 318.17,A -85,B 0,C 180,E1 -5805.47,E2 -5805.47} C_VEL
LIN {X 0,Y 502.827,Z 318.289,A -85,B 0,C 180,E1 -5808.806,E2 -5808.806} C_VEL
LIN {X 0,Y 506.726,Z 331.279,A -85,B 0,C 180,E1 -5811.612,E2 -5811.612} C_VEL
LIN {X 0,Y 509.813,Z 342.813,A -85,B 0,C 180,E1 -5813.888,E2 -5813.888} C_VEL
LIN {X 0,Y 509.611,Z 348.656,A -85,B 0,C 180,E1 -5814.85,E2 -5814.85} C_VEL
LIN {X 0,Y 508.481,Z 366.187,A -85,B 0,C 180,E1 -5817.603,E2 -5817.603} C_VEL
LIN {X 0,Y 507.526,Z 385.483,A -85,B 0,C 180,E1 -5820.51,E2 -5820.51} C_VEL
LIN {X 0,Y 506.617,Z 403.581,A -85,B 0,C 180,E1 -5823.204,E2 -5823.204} C_VEL
LIN {X 0,Y 505.84,Z 420.76,A -85,B 0,C 180,E1 -5825.717,E2 -5825.717} C_VEL
LIN {X 0,Y 509.864,Z 439.291,A -85,B 0,C 180,E1 -5826.22,E2 -5826.22} C_VEL
LIN {X 0,Y 509.408,Z 456.636,A -85,B 0,C 180,E1 -5826.615,E2 -5826.615} C_VEL
LIN {X 0,Y 508.866,Z 473.095,A -85,B 0,C 180,E1 -5827.162,E2 -5827.162} C_VEL
LIN {X 0,Y 508.243,Z 488.125,A -85,B 0,C 180,E1 -5827.811,E2 -5827.811} C_VEL
LIN {X 0,Y 507.461,Z 504.111,A -85,B 0,C 180,E1 -5828.687,E2 -5828.687} C_VEL
LIN {X 0,Y 506.599,Z 519.302,A -85,B 0,C 180,E1 -5829.709,E2 -5829.709} C_VEL
LIN {X 0,Y 505.748,Z 533.321,A -85,B 0,C 180,E1 -5830.844,E2 -5830.844} C_VEL
LIN {X 0,Y 504.94,Z 547.088,A -85,B 0,C 180,E1 -5832.172,E2 -5832.172} C_VEL
LIN {X 0,Y 504.314,Z 558.029,A -85,B 0,C 180,E1 -5833.403,E2 -5833.403} C_VEL
LIN {X 0,Y 503.788,Z 568.919,A -85,B 0,C 180,E1 -5834.839,E2 -5834.839} C_VEL
LIN {X 0,Y 503.208,Z 578.225,A -85,B 0,C 180,E1 -5836.267,E2 -5836.267} C_VEL
LIN {X 0,Y 502.849,Z 587.282,A -85,B 0,C 180,E1 -5837.901,E2 -5837.901} C_VEL
LIN {X 0,Y 502.514,Z 594.862,A -85,B 0,C 180,E1 -5839.527,E2 -5839.527} C_VEL
LIN {X 0,Y 502.303,Z 602.471,A -85,B 0,C 180,E1 -5841.554,E2 -5841.554} C_VEL
LIN {X 0,Y 502.181,Z 608.25,A -85,B 0,C 180,E1 -5843.574,E2 -5843.574} C_VEL
LIN {X 0,Y 502.06,Z 611.638,A -85,B 0,C 180,E1 -5845.184,E2 -5845.184} C_VEL
LIN {X 0,Y 502.102,Z 614.092,A -85,B 0,C 180,E1 -5846.792,E2 -5846.792} C_VEL
LIN {X 0,Y 502.03,Z 615.48,A -85,B 0,C 180,E1 -5848.398,E2 -5848.398} C_VEL
LIN {X 0,Y 501.975,Z 616,A -85,B 0,C 180,E1 -5850.002,E2 -5850.002} C_VEL
LIN {X 0,Y 502.03,Z 615.478,A -85,B 0,C 180,E1 -5851.606,E2 -5851.606} C_VEL
LIN {X 0,Y 502.103,Z 614.086,A -85,B 0,C 180,E1 -5853.211,E2 -5853.211} C_VEL
LIN {X 0,Y 502.062,Z 611.632,A -85,B 0,C 180,E1 -5854.82,E2 -5854.82} C_VEL
LIN {X 0,Y 502.185,Z 608.139,A -85,B 0,C 180,E1 -5856.471,E2 -5856.471} C_VEL
LIN {X 0,Y 502.298,Z 602.462,A -85,B 0,C 180,E1 -5858.45,E2 -5858.45} C_VEL
LIN {X 0,Y 502.516,Z 594.849,A -85,B 0,C 180,E1 -5860.477,E2 -5860.477} C_VEL
LIN {X 0,Y 502.883,Z 586.245,A -85,B 0,C 180,E1 -5862.307,E2 -5862.307} C_VEL
LIN {X 0,Y 503.282,Z 576.966,A -85,B 0,C 180,E1 -5863.94,E2 -5863.94} C_VEL
LIN {X 0,Y 503.815,Z 567.41,A -85,B 0,C 180,E1 -5865.371,E2 -5865.371} C_VEL
LIN {X 0,Y 504.417,Z 556.269,A -85,B 0,C 180,E1 -5866.806,E2 -5866.806} C_VEL
LIN {X 0,Y 505.139,Z 544.124,A -85,B 0,C 180,E1 -5868.139,E2 -5868.139} C_VEL
LIN {X 0,Y 505.924,Z 530.757,A -85,B 0,C 180,E1 -5869.379,E2 -5869.379} C_VEL
LIN {X 0,Y 506.704,Z 517.826,A -85,B 0,C 180,E1 -5870.396,E2 -5870.396} C_VEL
LIN {X 0,Y 507.448,Z 504.035,A -85,B 0,C 180,E1 -5871.318,E2 -5871.318} C_VEL
LIN {X 0,Y 508.242,Z 488.697,A -85,B 0,C 180,E1 -5872.158,E2 -5872.158} C_VEL
LIN {X 0,Y 508.854,Z 474.109,A -85,B 0,C 180,E1 -5872.797,E2 -5872.797} C_VEL
LIN {X 0,Y 509.412,Z 457.545,A -85,B 0,C 180,E1 -5873.358,E2 -5873.358} C_VEL
LIN {X 0,Y 509.83,Z 442.349,A -85,B 0,C 180,E1 -5873.727,E2 -5873.727} C_VEL
LIN {X 0,Y 509.657,Z 437.881,A -85,B 0,C 180,E1 -5873.815,E2 -5873.815} C_VEL
LIN {X 0,Y 505.841,Z 420.588,A -85,B 0,C 180,E1 -5874.308,E2 -5874.308} C_VEL
LIN {X 0,Y 506.627,Z 403.552,A -85,B 0,C 180,E1 -5876.799,E2 -5876.799} C_VEL
LIN {X 0,Y 507.619,Z 382.804,A -85,B 0,C 180,E1 -5879.897,E2 -5879.897} C_VEL
LIN {X 0,Y 508.573,Z 364.673,A -85,B 0,C 180,E1 -5882.613,E2 -5882.613} C_VEL
LIN {X 0,Y 509.226,Z 354.691,A -85,B 0,C 180,E1 -5884.195,E2 -5884.195} C_VEL
LIN {X 0,Y 510.095,Z 344.67,A -85,B 0,C 180,E1 -5885.868,E2 -5885.868} C_VEL
LIN {X 0,Y 509.27,Z 339.923,A -85,B 0,C 180,E1 -5886.831,E2 -5886.831} C_VEL
LIN {X 0,Y 507.535,Z 333.323,A -85,B 0,C 180,E1 -5888.379,E2 -5888.379} C_VEL
LIN {X 0,Y 505.634,Z 327.194,A -85,B 0,C 180,E1 -5890.141,E2 -5890.141} C_VEL
LIN {X 0,Y 503.985,Z 322.149,A -85,B 0,C 180,E1 -5892.019,E2 -5892.019} C_VEL
LIN {X 0,Y 502.835,Z 318.599,A -85,B 0,C 180,E1 -5893.899,E2 -5893.899} C_VEL
LIN {X 0,Y 502.783,Z 318.173,A -85,B 0,C 180,E1 -5894.341,E2 -5894.341} C_VEL
LIN {X 0,Y 502.759,Z 318.175,A -85,B 0,C 180,E1 -5896.768,E2 -5896.768} C_VEL
LIN {X 0,Y 502.78,Z 318.173,A -85,B 0,C 180,E1 -5899.012,E2 -5899.012} C_VEL
LIN {X 0,Y 502.779,Z 318.217,A -85,B 0,C 180,E1 -5900.248,E2 -5900.248} C_VEL
LIN {X 0,Y 503.383,Z 320.856,A -85,B 0,C 180,E1 -5902.099,E2 -5902.099} C_VEL
LIN {X 0,Y 504.161,Z 324.48,A -85,B 0,C 180,E1 -5904.163,E2 -5904.163} C_VEL
LIN {X 0,Y 504.22,Z 328.372,A -85,B 0,C 180,E1 -5906.115,E2 -5906.115} C_VEL
LIN {X 0,Y 503.889,Z 334.194,A -85,B 0,C 180,E1 -5908.932,E2 -5908.932} C_VEL
LIN {X 0,Y 503.694,Z 339.647,A -85,B 0,C 180,E1 -5911.68,E2 -5911.68} C_VEL
LIN {X 0,Y 503.548,Z 344.88,A -85,B 0,C 180,E1 -5914.363,E2 -5914.363} C_VEL
LIN {X 0,Y 503.359,Z 350.201,A -85,B 0,C 180,E1 -5917.149,E2 -5917.149} C_VEL
LIN {X 0,Y 503.218,Z 354.774,A -85,B 0,C 180,E1 -5919.565,E2 -5919.565} C_VEL
LIN {X 0,Y 503.041,Z 359.587,A -85,B 0,C 180,E1 -5922.1,E2 -5922.1} C_VEL
LIN {X 0,Y 502.886,Z 365.916,A -85,B 0,C 180,E1 -5925.406,E2 -5925.406} C_VEL
LIN {X 0,Y 505.622,Z 375.427,A -85,B 0,C 180,E1 -5925.8,E2 -5925.8} C_VEL
LIN {X 0,Y 505.374,Z 389.156,A -85,B 0,C 180,E1 -5926.325,E2 -5926.325} C_VEL
LIN {X 0,Y 504.927,Z 401.95,A -85,B 0,C 180,E1 -5926.99,E2 -5926.99} C_VEL
LIN {X 0,Y 504.543,Z 413.889,A -85,B 0,C 180,E1 -5927.796,E2 -5927.796} C_VEL
LIN {X 0,Y 504.135,Z 425.092,A -85,B 0,C 180,E1 -5928.746,E2 -5928.746} C_VEL
LIN {X 0,Y 503.838,Z 434.65,A -85,B 0,C 180,E1 -5929.756,E2 -5929.756} C_VEL
LIN {X 0,Y 503.456,Z 443.974,A -85,B 0,C 180,E1 -5930.965,E2 -5930.965} C_VEL
LIN {X 0,Y 503.182,Z 451.528,A -85,B 0,C 180,E1 -5932.194,E2 -5932.194} C_VEL
LIN {X 0,Y 502.89,Z 458.256,A -85,B 0,C 180,E1 -5933.581,E2 -5933.581} C_VEL
LIN {X 0,Y 502.694,Z 462.795,A -85,B 0,C 180,E1 -5934.786,E2 -5934.786} C_VEL
LIN {X 0,Y 502.695,Z 466.224,A -85,B 0,C 180,E1 -5935.992,E2 -5935.992} C_VEL
LIN {X 0,Y 502.606,Z 467.991,A -85,B 0,C 180,E1 -5936.794,E2 -5936.794} C_VEL
LIN {X 0,Y 502.528,Z 469.324,A -85,B 0,C 180,E1 -5937.596,E2 -5937.596} C_VEL
LIN {X 0,Y 502.424,Z 470.258,A -85,B 0,C 180,E1 -5938.397,E2 -5938.397} C_VEL
LIN {X 0,Y 502.356,Z 470.93,A -85,B 0,C 180,E1 -5940,E2 -5940} C_VEL
LIN {X 0,Y 502.42,Z 470.035,A -85,B 0,C 180,E1 -5941.603,E2 -5941.603} C_VEL
LIN {X 0,Y 502.43,Z 468.988,A -85,B 0,C 180,E1 -5942.405,E2 -5942.405} C_VEL
LIN {X 0,Y 502.52,Z 467.533,A -85,B 0,C 180,E1 -5943.207,E2 -5943.207} C_VEL
LIN {X 0,Y 502.517,Z 464.577,A -85,B 0,C 180,E1 -5944.412,E2 -5944.412} C_VEL
LIN {X 0,Y 502.583,Z 460.598,A -85,B 0,C 180,E1 -5945.618,E2 -5945.618} C_VEL
LIN {X 0,Y 502.762,Z 454.547,A -85,B 0,C 180,E1 -5947.019,E2 -5947.019} C_VEL
LIN {X 0,Y 502.993,Z 447.863,A -85,B 0,C 180,E1 -5948.234,E2 -5948.234} C_VEL
LIN {X 0,Y 503.224,Z 439.581,A -85,B 0,C 180,E1 -5949.445,E2 -5949.445} C_VEL
LIN {X 0,Y 503.468,Z 431.148,A -85,B 0,C 180,E1 -5950.456,E2 -5950.456} C_VEL
LIN {X 0,Y 503.841,Z 420.822,A -85,B 0,C 180,E1 -5951.465,E2 -5951.465} C_VEL
LIN {X 0,Y 504.167,Z 409.53,A -85,B 0,C 180,E1 -5952.354,E2 -5952.354} C_VEL
LIN {X 0,Y 504.557,Z 397.853,A -85,B 0,C 180,E1 -5953.082,E2 -5953.082} C_VEL
LIN {X 0,Y 504.822,Z 385.141,A -85,B 0,C 180,E1 -5953.69,E2 -5953.69} C_VEL
LIN {X 0,Y 504.915,Z 374.55,A -85,B 0,C 180,E1 -5954.073,E2 -5954.073} C_VEL
LIN {X 0,Y 502.685,Z 364.414,A -85,B 0,C 180,E1 -5954.417,E2 -5954.417} C_VEL
LIN {X 0,Y 502.372,Z 362.871,A -85,B 0,C 180,E1 -5954.482,E2 -5954.482} C_VEL
LIN {X 0,Y 502.402,Z 357.478,A -85,B 0,C 180,E1 -5957.084,E2 -5957.084} C_VEL
LIN {X 0,Y 502.478,Z 352.264,A -85,B 0,C 180,E1 -5959.614,E2 -5959.614} C_VEL
LIN {X 0,Y 502.674,Z 346.032,A -85,B 0,C 180,E1 -5962.665,E2 -5962.665} C_VEL
LIN {X 0,Y 502.732,Z 339.953,A -85,B 0,C 180,E1 -5965.682,E2 -5965.682} C_VEL
LIN {X 0,Y 502.862,Z 334.533,A -85,B 0,C 180,E1 -5968.372,E2 -5968.372} C_VEL
LIN {X 0,Y 502.946,Z 329.027,A -85,B 0,C 180,E1 -5971.133,E2 -5971.133} C_VEL
LIN {X 0,Y 503.085,Z 323.395,A -85,B 0,C 180,E1 -5973.973,E2 -5973.973} C_VEL
LIN {X 0,Y 502.866,Z 318.346,A -85,B 0,C 180,E1 -5976.565,E2 -5976.565} C_VEL
LIN {X 0,Y 502.791,Z 318.171,A -85,B 0,C 180,E1 -5979.753,E2 -5979.753} C_VEL
LIN {X 0,Y 502.812,Z 318.166,A -85,B 0,C 180,E1 -5982.199,E2 -5982.199} C_VEL
LIN {X 0,Y 502.794,Z 318.17,A -85,B 0,C 180,E1 -5985.47,E2 -5985.47} C_VEL
LIN {X 0,Y 502.787,Z 318.169,A -85,B 0,C 180,E1 -5988.162,E2 -5988.162} C_VEL
LIN {X 0,Y 502.805,Z 318.168,A -85,B 0,C 180,E1 -5991.023,E2 -5991.023} C_VEL
LIN {X 0,Y 502.796,Z 318.17,A -85,B 0,C 180,E1 -5991.648,E2 -5991.648} C_VEL
LIN {X 0,Y 502.112,Z 318.256,A -85,B 0,C 180,E1 -5992.099,E2 -5992.099} C_VEL
LIN {X 0,Y 496.502,Z 319.207,A -85,B 0,C 180,E1 -5993.508,E2 -5993.508} C_VEL
LIN {X 0,Y 495.942,Z 320.04,A -85,B 0,C 180,E1 -5993.951,E2 -5993.951} C_VEL
LIN {X 0,Y 496.274,Z 323.852,A -85,B 0,C 180,E1 -5995.495,E2 -5995.495} C_VEL
LIN {X 0,Y 496.236,Z 328.429,A -85,B 0,C 180,E1 -5997.439,E2 -5997.439} C_VEL
LIN {X 0,Y 496.165,Z 334.606,A -85,B 0,C 180,E1 -6000.278,E2 -6000.278} C_VEL
LIN {X 0,Y 496.033,Z 340.599,A -85,B 0,C 180,E1 -6003.204,E2 -6003.204} C_VEL
LIN {X 0,Y 495.958,Z 345.644,A -85,B 0,C 180,E1 -6005.734,E2 -6005.734} C_VEL
LIN {X 0,Y 495.838,Z 350.947,A -85,B 0,C 180,E1 -6008.374,E2 -6008.374} C_VEL
LIN {X 0,Y 495.765,Z 356.411,A -85,B 0,C 180,E1 -6010.969,E2 -6010.969} C_VEL
LIN {X 0,Y 495.758,Z 362.162,A -85,B 0,C 180,E1 -6013.528,E2 -6013.528} C_VEL
LIN {X 0,Y 495.829,Z 367.042,A -85,B 0,C 180,E1 -6015.571,E2 -6015.571} C_VEL
LIN {X 0,Y 498.139,Z 375.974,A -85,B 0,C 180,E1 -6015.851,E2 -6015.851} C_VEL
LIN {X 0,Y 497.982,Z 388.433,A -85,B 0,C 180,E1 -6016.273,E2 -6016.273} C_VEL
LIN {X 0,Y 497.723,Z 400.307,A -85,B 0,C 180,E1 -6016.837,E2 -6016.837} C_VEL
LIN {X 0,Y 497.504,Z 411.592,A -85,B 0,C 180,E1 -6017.542,E2 -6017.542} C_VEL
LIN {X 0,Y 497.154,Z 422.177,A -85,B 0,C 180,E1 -6018.377,E2 -6018.377} C_VEL
LIN {X 0,Y 496.766,Z 432.506,A -85,B 0,C 180,E1 -6019.4,E2 -6019.4} C_VEL
LIN {X 0,Y 496.488,Z 440.906,A -85,B 0,C 180,E1 -6020.424,E2 -6020.424} C_VEL
LIN {X 0,Y 496.125,Z 449.09,A -85,B 0,C 180,E1 -6021.649,E2 -6021.649} C_VEL
LIN {X 0,Y 495.881,Z 455.23,A -85,B 0,C 180,E1 -6022.793,E2 -6022.793} C_VEL
LIN {X 0,Y 495.774,Z 460.037,A -85,B 0,C 180,E1 -6023.895,E2 -6023.895} C_VEL
LIN {X 0,Y 495.525,Z 464.286,A -85,B 0,C 180,E1 -6025.116,E2 -6025.116} C_VEL
LIN {X 0,Y 495.51,Z 466.503,A -85,B 0,C 180,E1 -6025.931,E2 -6025.931} C_VEL
LIN {X 0,Y 495.454,Z 468.318,A -85,B 0,C 180,E1 -6026.745,E2 -6026.745} C_VEL
LIN {X 0,Y 495.427,Z 469.706,A -85,B 0,C 180,E1 -6027.559,E2 -6027.559} C_VEL
LIN {X 0,Y 495.363,Z 471.282,A -85,B 0,C 180,E1 -6029.185,E2 -6029.185} C_VEL
LIN {X 0,Y 495.35,Z 471.516,A -85,B 0,C 180,E1 -6029.998,E2 -6029.998} C_VEL
LIN {X 0,Y 495.362,Z 471.335,A -85,B 0,C 180,E1 -6030.811,E2 -6030.811} C_VEL
LIN {X 0,Y 495.432,Z 469.827,A -85,B 0,C 180,E1 -6032.437,E2 -6032.437} C_VEL
LIN {X 0,Y 495.539,Z 468.495,A -85,B 0,C 180,E1 -6033.25,E2 -6033.25} C_VEL
LIN {X 0,Y 495.599,Z 465.711,A -85,B 0,C 180,E1 -6034.471,E2 -6034.471} C_VEL
LIN {X 0,Y 495.679,Z 461.926,A -85,B 0,C 180,E1 -6035.694,E2 -6035.694} C_VEL
LIN {X 0,Y 495.816,Z 455.939,A -85,B 0,C 180,E1 -6037.148,E2 -6037.148} C_VEL
LIN {X 0,Y 496.117,Z 449.62,A -85,B 0,C 180,E1 -6038.347,E2 -6038.347} C_VEL
LIN {X 0,Y 496.462,Z 441.617,A -85,B 0,C 180,E1 -6039.573,E2 -6039.573} C_VEL
LIN {X 0,Y 496.759,Z 433.362,A -85,B 0,C 180,E1 -6040.596,E2 -6040.596} C_VEL
LIN {X 0,Y 497.099,Z 423.202,A -85,B 0,C 180,E1 -6041.62,E2 -6041.62} C_VEL
LIN {X 0,Y 497.471,Z 413.019,A -85,B 0,C 180,E1 -6042.447,E2 -6042.447} C_VEL
LIN {X 0,Y 497.697,Z 402.006,A -85,B 0,C 180,E1 -6043.159,E2 -6043.159} C_VEL
LIN {X 0,Y 497.985,Z 389.413,A -85,B 0,C 180,E1 -6043.775,E2 -6043.775} C_VEL
LIN {X 0,Y 498.143,Z 376.928,A -85,B 0,C 180,E1 -6044.213,E2 -6044.213} C_VEL
LIN {X 0,Y 497.23,Z 372.028,A -85,B 0,C 180,E1 -6044.371,E2 -6044.371} C_VEL
LIN {X 0,Y 495.811,Z 367.034,A -85,B 0,C 180,E1 -6044.531,E2 -6044.531} C_VEL
LIN {X 0,Y 495.73,Z 360.429,A -85,B 0,C 180,E1 -6047.318,E2 -6047.318} C_VEL
LIN {X 0,Y 495.834,Z 353.074,A -85,B 0,C 180,E1 -6050.691,E2 -6050.691} C_VEL
LIN {X 0,Y 495.906,Z 347.629,A -85,B 0,C 180,E1 -6053.377,E2 -6053.377} C_VEL
LIN {X 0,Y 496.012,Z 342.283,A -85,B 0,C 180,E1 -6056.053,E2 -6056.053} C_VEL
LIN {X 0,Y 496.092,Z 336.759,A -85,B 0,C 180,E1 -6058.792,E2 -6058.792} C_VEL
LIN {X 0,Y 496.2,Z 330.799,A -85,B 0,C 180,E1 -6061.601,E2 -6061.601} C_VEL
LIN {X 0,Y 496.297,Z 325.325,A -85,B 0,C 180,E1 -6064.008,E2 -6064.008} C_VEL
LIN {X 0,Y 496.219,Z 321.68,A -85,B 0,C 180,E1 -6065.496,E2 -6065.496} C_VEL
LIN {X 0,Y 495.784,Z 319.046,A -85,B 0,C 180,E1 -6066.536,E2 -6066.536} C_VEL
LIN {X 0,Y 495.744,Z 319.048,A -85,B 0,C 180,E1 -6069.635,E2 -6069.635} C_VEL
LIN {X 0,Y 495.72,Z 319.048,A -85,B 0,C 180,E1 -6072.504,E2 -6072.504} C_VEL
LIN {X 0,Y 495.734,Z 319.05,A -85,B 0,C 180,E1 -6075.137,E2 -6075.137} C_VEL
LIN {X 0,Y 495.77,Z 319.041,A -85,B 0,C 180,E1 -6078.22,E2 -6078.22} C_VEL
LIN {X 0,Y 495.765,Z 319.041,A -85,B 0,C 180,E1 -6081.227,E2 -6081.227} C_VEL
LIN {X 0,Y 495.737,Z 319.045,A -85,B 0,C 180,E1 -6084.461,E2 -6084.461} C_VEL
LIN {X 0,Y 495.747,Z 319.047,A -85,B 0,C 180,E1 -6087.404,E2 -6087.404} C_VEL
LIN {X 0,Y 495.745,Z 319.041,A -85,B 0,C 180,E1 -6090.252,E2 -6090.252} C_VEL
LIN {X 0,Y 495.813,Z 319.032,A -85,B 0,C 180,E1 -6093.247,E2 -6093.247} C_VEL
LIN {X 0,Y 495.752,Z 319.044,A -85,B 0,C 180,E1 -6095.725,E2 -6095.725} C_VEL
LIN {X 0,Y 495.745,Z 319.044,A -85,B 0,C 180,E1 -6098.371,E2 -6098.371} C_VEL
LIN {X 0,Y 495.76,Z 319.041,A -85,B 0,C 180,E1 -6100.97,E2 -6100.97} C_VEL
LIN {X 0,Y 495.754,Z 319.044,A -85,B 0,C 180,E1 -6103.529,E2 -6103.529} C_VEL
LIN {X 0,Y 495.773,Z 319.035,A -85,B 0,C 180,E1 -6106.055,E2 -6106.055} C_VEL
LIN {X 0,Y 495.857,Z 319.032,A -85,B 0,C 180,E1 -6108.555,E2 -6108.555} C_VEL
LIN {X 0,Y 495.855,Z 319.032,A -85,B 0,C 180,E1 -6111.851,E2 -6111.851} C_VEL
LIN {X 0,Y 495.88,Z 319.024,A -85,B 0,C 180,E1 -6114.306,E2 -6114.306} C_VEL
LIN {X 0,Y 495.963,Z 319.018,A -85,B 0,C 180,E1 -6117.563,E2 -6117.563} C_VEL
LIN {X 0,Y 495.969,Z 319.013,A -85,B 0,C 180,E1 -6120,E2 -6120} C_VEL
LIN {X 0,Y 495.975,Z 319.019,A -85,B 0,C 180,E1 -6122.436,E2 -6122.436} C_VEL
LIN {X 0,Y 495.896,Z 319.029,A -85,B 0,C 180,E1 -6125.693,E2 -6125.693} C_VEL
LIN {X 0,Y 495.849,Z 319.031,A -85,B 0,C 180,E1 -6128.148,E2 -6128.148} C_VEL
LIN {X 0,Y 495.849,Z 319.033,A -85,B 0,C 180,E1 -6131.445,E2 -6131.445} C_VEL
LIN {X 0,Y 495.767,Z 319.045,A -85,B 0,C 180,E1 -6134.783,E2 -6134.783} C_VEL
LIN {X 0,Y 495.777,Z 319.039,A -85,B 0,C 180,E1 -6137.319,E2 -6137.319} C_VEL
LIN {X 0,Y 495.755,Z 319.047,A -85,B 0,C 180,E1 -6139.891,E2 -6139.891} C_VEL
LIN {X 0,Y 495.765,Z 319.042,A -85,B 0,C 180,E1 -6142.87,E2 -6142.87} C_VEL
LIN {X 0,Y 495.766,Z 319.04,A -85,B 0,C 180,E1 -6146.069,E2 -6146.069} C_VEL
LIN {X 0,Y 495.747,Z 319.046,A -85,B 0,C 180,E1 -6148.816,E2 -6148.816} C_VEL
LIN {X 0,Y 495.737,Z 319.048,A -85,B 0,C 180,E1 -6151.727,E2 -6151.727} C_VEL
LIN {X 0,Y 495.756,Z 319.043,A -85,B 0,C 180,E1 -6154.697,E2 -6154.697} C_VEL
LIN {X 0,Y 495.713,Z 319.05,A -85,B 0,C 180,E1 -6157.563,E2 -6157.563} C_VEL
LIN {X 0,Y 495.746,Z 319.048,A -85,B 0,C 180,E1 -6160.702,E2 -6160.702} C_VEL
LIN {X 0,Y 495.714,Z 319.047,A -85,B 0,C 180,E1 -6164.003,E2 -6164.003} C_VEL
LIN {X 0,Y 495.746,Z 319.05,A -85,B 0,C 180,E1 -6167.123,E2 -6167.123} C_VEL
LIN {X 0,Y 495.816,Z 319.195,A -85,B 0,C 180,E1 -6168.229,E2 -6168.229} C_VEL
LIN {X 0,Y 499.537,Z 331.732,A -85,B 0,C 180,E1 -6171.015,E2 -6171.015} C_VEL
LIN {X 0,Y 502.263,Z 341.42,A -85,B 0,C 180,E1 -6173.013,E2 -6173.013} C_VEL
LIN {X 0,Y 503.308,Z 345.759,A -85,B 0,C 180,E1 -6173.849,E2 -6173.849} C_VEL
LIN {X 0,Y 502.218,Z 361.743,A -85,B 0,C 180,E1 -6176.447,E2 -6176.447} C_VEL
LIN {X 0,Y 501.281,Z 377.733,A -85,B 0,C 180,E1 -6178.924,E2 -6178.924} C_VEL
LIN {X 0,Y 500.397,Z 394.689,A -85,B 0,C 180,E1 -6181.479,E2 -6181.479} C_VEL
LIN {X 0,Y 499.312,Z 415.816,A -85,B 0,C 180,E1 -6184.637,E2 -6184.637} C_VEL
LIN {X 0,Y 499.068,Z 420.712,A -85,B 0,C 180,E1 -6185.359,E2 -6185.359} C_VEL
LIN {X 0,Y 503.384,Z 440.366,A -85,B 0,C 180,E1 -6185.914,E2 -6185.914} C_VEL
LIN {X 0,Y 502.869,Z 457.113,A -85,B 0,C 180,E1 -6186.307,E2 -6186.307} C_VEL
LIN {X 0,Y 502.279,Z 474.261,A -85,B 0,C 180,E1 -6186.894,E2 -6186.894} C_VEL
LIN {X 0,Y 501.584,Z 489.169,A -85,B 0,C 180,E1 -6187.557,E2 -6187.557} C_VEL
LIN {X 0,Y 500.8,Z 504.285,A -85,B 0,C 180,E1 -6188.4,E2 -6188.4} C_VEL
LIN {X 0,Y 499.912,Z 519.302,A -85,B 0,C 180,E1 -6189.426,E2 -6189.426} C_VEL
LIN {X 0,Y 499.095,Z 532.383,A -85,B 0,C 180,E1 -6190.493,E2 -6190.493} C_VEL
LIN {X 0,Y 498.226,Z 545.142,A -85,B 0,C 180,E1 -6191.711,E2 -6191.711} C_VEL
LIN {X 0,Y 497.532,Z 556.299,A -85,B 0,C 180,E1 -6192.958,E2 -6192.958} C_VEL
LIN {X 0,Y 496.895,Z 567.438,A -85,B 0,C 180,E1 -6194.414,E2 -6194.414} C_VEL
LIN {X 0,Y 496.237,Z 578.224,A -85,B 0,C 180,E1 -6196.071,E2 -6196.071} C_VEL
LIN {X 0,Y 495.81,Z 587.282,A -85,B 0,C 180,E1 -6197.726,E2 -6197.726} C_VEL
LIN {X 0,Y 495.471,Z 594.861,A -85,B 0,C 180,E1 -6199.376,E2 -6199.376} C_VEL
LIN {X 0,Y 495.215,Z 602.471,A -85,B 0,C 180,E1 -6201.432,E2 -6201.432} C_VEL
LIN {X 0,Y 495.099,Z 608.25,A -85,B 0,C 180,E1 -6203.482,E2 -6203.482} C_VEL
LIN {X 0,Y 494.983,Z 611.638,A -85,B 0,C 180,E1 -6205.115,E2 -6205.115} C_VEL
LIN {X 0,Y 495.022,Z 614.092,A -85,B 0,C 180,E1 -6206.747,E2 -6206.747} C_VEL
LIN {X 0,Y 494.955,Z 615.48,A -85,B 0,C 180,E1 -6208.375,E2 -6208.375} C_VEL
LIN {X 0,Y 494.893,Z 616,A -85,B 0,C 180,E1 -6210.002,E2 -6210.002} C_VEL
LIN {X 0,Y 494.956,Z 615.477,A -85,B 0,C 180,E1 -6211.629,E2 -6211.629} C_VEL
LIN {X 0,Y 495.023,Z 614.087,A -85,B 0,C 180,E1 -6213.257,E2 -6213.257} C_VEL
LIN {X 0,Y 494.984,Z 611.631,A -85,B 0,C 180,E1 -6214.889,E2 -6214.889} C_VEL
LIN {X 0,Y 495.103,Z 608.246,A -85,B 0,C 180,E1 -6216.522,E2 -6216.522} C_VEL
LIN {X 0,Y 495.208,Z 602.462,A -85,B 0,C 180,E1 -6218.572,E2 -6218.572} C_VEL
LIN {X 0,Y 495.473,Z 594.849,A -85,B 0,C 180,E1 -6220.628,E2 -6220.628} C_VEL
LIN {X 0,Y 495.854,Z 586.246,A -85,B 0,C 180,E1 -6222.485,E2 -6222.485} C_VEL
LIN {X 0,Y 496.312,Z 576.967,A -85,B 0,C 180,E1 -6224.14,E2 -6224.14} C_VEL
LIN {X 0,Y 496.86,Z 567.409,A -85,B 0,C 180,E1 -6225.592,E2 -6225.592} C_VEL
LIN {X 0,Y 497.539,Z 556.269,A -85,B 0,C 180,E1 -6227.046,E2 -6227.046} C_VEL
LIN {X 0,Y 498.295,Z 544.124,A -85,B 0,C 180,E1 -6228.397,E2 -6228.397} C_VEL
LIN {X 0,Y 499.152,Z 530.932,A -85,B 0,C 180,E1 -6229.637,E2 -6229.637} C_VEL
LIN {X 0,Y 500.008,Z 517.824,A -85,B 0,C 180,E1 -6230.682,E2 -6230.682} C_VEL
LIN {X 0,Y 500.794,Z 504.207,A -85,B 0,C 180,E1 -6231.605,E2 -6231.605} C_VEL
LIN {X 0,Y 501.683,Z 488.384,A -85,B 0,C 180,E1 -6232.481,E2 -6232.481} C_VEL
LIN {X 0,Y 502.285,Z 474.173,A -85,B 0,C 180,E1 -6233.11,E2 -6233.11} C_VEL
LIN {X 0,Y 502.872,Z 458.027,A -85,B 0,C 180,E1 -6233.666,E2 -6233.666} C_VEL
LIN {X 0,Y 503.361,Z 442.165,A -85,B 0,C 180,E1 -6234.054,E2 -6234.054} C_VEL
LIN {X 0,Y 502.927,Z 438.025,A -85,B 0,C 180,E1 -6234.152,E2 -6234.152} C_VEL
LIN {X 0,Y 499.054,Z 420.602,A -85,B 0,C 180,E1 -6234.658,E2 -6234.658} C_VEL
LIN {X 0,Y 499.848,Z 405.034,A -85,B 0,C 180,E1 -6236.966,E2 -6236.966} C_VEL
LIN {X 0,Y 500.862,Z 385.758,A -85,B 0,C 180,E1 -6239.877,E2 -6239.877} C_VEL
LIN {X 0,Y 501.95,Z 364.23,A -85,B 0,C 180,E1 -6243.098,E2 -6243.098} C_VEL
LIN {X 0,Y 503.459,Z 347.461,A -85,B 0,C 180,E1 -6245.939,E2 -6245.939} C_VEL
LIN {X 0,Y 503.025,Z 343.78,A -85,B 0,C 180,E1 -6246.677,E2 -6246.677} C_VEL
LIN {X 0,Y 501.34,Z 336.985,A -85,B 0,C 180,E1 -6248.277,E2 -6248.277} C_VEL
LIN {X 0,Y 499.586,Z 331.152,A -85,B 0,C 180,E1 -6249.944,E2 -6249.944} C_VEL
LIN {X 0,Y 498.082,Z 326.515,A -85,B 0,C 180,E1 -6251.597,E2 -6251.597} C_VEL
LIN {X 0,Y 497.224,Z 324.029,A -85,B 0,C 180,E1 -6252.724,E2 -6252.724} C_VEL
LIN {X 0,Y 496.597,Z 321.967,A -85,B 0,C 180,E1 -6253.906,E2 -6253.906} C_VEL
LIN {X 0,Y 496.08,Z 320.536,A -85,B 0,C 180,E1 -6255.103,E2 -6255.103} C_VEL
LIN {X 0,Y 495.834,Z 319.661,A -85,B 0,C 180,E1 -6256.294,E2 -6256.294} C_VEL
LIN {X 0,Y 495.817,Z 319.574,A -85,B 0,C 180,E1 -6258.226,E2 -6258.226} C_VEL
LIN {X 0,Y 496.288,Z 321.146,A -85,B 0,C 180,E1 -6260.413,E2 -6260.413} C_VEL
LIN {X 0,Y 496.904,Z 324.026,A -85,B 0,C 180,E1 -6262.543,E2 -6262.543} C_VEL
LIN {X 0,Y 497.439,Z 327.512,A -85,B 0,C 180,E1 -6264.602,E2 -6264.602} C_VEL
LIN {X 0,Y 497.347,Z 331.307,A -85,B 0,C 180,E1 -6266.557,E2 -6266.557} C_VEL
LIN {X 0,Y 496.982,Z 337.34,A -85,B 0,C 180,E1 -6269.614,E2 -6269.614} C_VEL
LIN {X 0,Y 496.692,Z 343.979,A -85,B 0,C 180,E1 -6273.055,E2 -6273.055} C_VEL
LIN {X 0,Y 496.522,Z 349.111,A -85,B 0,C 180,E1 -6275.765,E2 -6275.765} C_VEL
LIN {X 0,Y 496.338,Z 355.688,A -85,B 0,C 180,E1 -6279.269,E2 -6279.269} C_VEL
LIN {X 0,Y 496.038,Z 362.158,A -85,B 0,C 180,E1 -6282.691,E2 -6282.691} C_VEL
LIN {X 0,Y 495.951,Z 366.849,A -85,B 0,C 180,E1 -6285.141,E2 -6285.141} C_VEL
LIN {X 0,Y 499.006,Z 376.986,A -85,B 0,C 180,E1 -6285.575,E2 -6285.575} C_VEL
LIN {X 0,Y 498.666,Z 390.011,A -85,B 0,C 180,E1 -6286.086,E2 -6286.086} C_VEL
LIN {X 0,Y 498.213,Z 402.541,A -85,B 0,C 180,E1 -6286.744,E2 -6286.744} C_VEL
LIN {X 0,Y 497.768,Z 415.238,A -85,B 0,C 180,E1 -6287.614,E2 -6287.614} C_VEL
LIN {X 0,Y 497.317,Z 426.496,A -85,B 0,C 180,E1 -6288.589,E2 -6288.589} C_VEL
LIN {X 0,Y 496.979,Z 435.999,A -85,B 0,C 180,E1 -6289.613,E2 -6289.613} C_VEL
LIN {X 0,Y 496.567,Z 445.285,A -85,B 0,C 180,E1 -6290.839,E2 -6290.839} C_VEL
LIN {X 0,Y 496.28,Z 452.81,A -85,B 0,C 180,E1 -6292.084,E2 -6292.084} C_VEL
LIN {X 0,Y 495.95,Z 459.529,A -85,B 0,C 180,E1 -6293.491,E2 -6293.491} C_VEL
LIN {X 0,Y 495.747,Z 464.054,A -85,B 0,C 180,E1 -6294.713,E2 -6294.713} C_VEL
LIN {X 0,Y 495.726,Z 467.472,A -85,B 0,C 180,E1 -6295.935,E2 -6295.935} C_VEL
LIN {X 0,Y 495.649,Z 469.227,A -85,B 0,C 180,E1 -6296.749,E2 -6296.749} C_VEL
LIN {X 0,Y 495.548,Z 470.554,A -85,B 0,C 180,E1 -6297.562,E2 -6297.562} C_VEL
LIN {X 0,Y 495.373,Z 471.983,A -85,B 0,C 180,E1 -6299.187,E2 -6299.187} C_VEL
LIN {X 0,Y 495.357,Z 472.114,A -85,B 0,C 180,E1 -6300,E2 -6300} C_VEL
LIN {X 0,Y 495.368,Z 471.847,A -85,B 0,C 180,E1 -6300.813,E2 -6300.813} C_VEL
LIN {X 0,Y 495.426,Z 471.173,A -85,B 0,C 180,E1 -6301.626,E2 -6301.626} C_VEL
LIN {X 0,Y 495.535,Z 468.627,A -85,B 0,C 180,E1 -6303.252,E2 -6303.252} C_VEL
LIN {X 0,Y 495.515,Z 465.635,A -85,B 0,C 180,E1 -6304.474,E2 -6304.474} C_VEL
LIN {X 0,Y 495.598,Z 461.611,A -85,B 0,C 180,E1 -6305.697,E2 -6305.697} C_VEL
LIN {X 0,Y 495.798,Z 455.471,A -85,B 0,C 180,E1 -6307.128,E2 -6307.128} C_VEL
LIN {X 0,Y 496.04,Z 448.774,A -85,B 0,C 180,E1 -6308.351,E2 -6308.351} C_VEL
LIN {X 0,Y 496.282,Z 440.449,A -85,B 0,C 180,E1 -6309.579,E2 -6309.579} C_VEL
LIN {X 0,Y 496.55,Z 431.98,A -85,B 0,C 180,E1 -6310.603,E2 -6310.603} C_VEL
LIN {X 0,Y 496.939,Z 421.63,A -85,B 0,C 180,E1 -6311.627,E2 -6311.627} C_VEL
LIN {X 0,Y 497.283,Z 410.467,A -85,B 0,C 180,E1 -6312.517,E2 -6312.517} C_VEL
LIN {X 0,Y 497.712,Z 398.654,A -85,B 0,C 180,E1 -6313.266,E2 -6313.266} C_VEL
LIN {X 0,Y 497.979,Z 386.043,A -85,B 0,C 180,E1 -6313.882,E2 -6313.882} C_VEL
LIN {X 0,Y 498.028,Z 375.201,A -85,B 0,C 180,E1 -6314.285,E2 -6314.285} C_VEL
LIN {X 0,Y 495.347,Z 363.287,A -85,B 0,C 180,E1 -6314.692,E2 -6314.692} C_VEL
LIN {X 0,Y 495.372,Z 357.823,A -85,B 0,C 180,E1 -6317.334,E2 -6317.334} C_VEL
LIN {X 0,Y 495.494,Z 351.197,A -85,B 0,C 180,E1 -6320.586,E2 -6320.586} C_VEL
LIN {X 0,Y 495.601,Z 345.52,A -85,B 0,C 180,E1 -6323.395,E2 -6323.395} C_VEL
LIN {X 0,Y 495.704,Z 340.142,A -85,B 0,C 180,E1 -6326.073,E2 -6326.073} C_VEL
LIN {X 0,Y 495.855,Z 334.684,A -85,B 0,C 180,E1 -6328.81,E2 -6328.81} C_VEL
LIN {X 0,Y 495.965,Z 328.848,A -85,B 0,C 180,E1 -6331.763,E2 -6331.763} C_VEL
LIN {X 0,Y 496.085,Z 322.999,A -85,B 0,C 180,E1 -6334.745,E2 -6334.745} C_VEL
LIN {X 0,Y 495.786,Z 319.043,A -85,B 0,C 180,E1 -6336.856,E2 -6336.856} C_VEL
LIN {X 0,Y 495.764,Z 319.048,A -85,B 0,C 180,E1 -6340.046,E2 -6340.046} C_VEL
LIN {X 0,Y 495.725,Z 319.05,A -85,B 0,C 180,E1 -6342.884,E2 -6342.884} C_VEL
LIN {X 0,Y 495.732,Z 319.049,A -85,B 0,C 180,E1 -6345.997,E2 -6345.997} C_VEL
LIN {X 0,Y 495.748,Z 319.047,A -85,B 0,C 180,E1 -6348.709,E2 -6348.709} C_VEL
LIN {X 0,Y 495.737,Z 319.049,A -85,B 0,C 180,E1 -6351.643,E2 -6351.643} C_VEL
LIN {X 0,Y 495.798,Z 319.094,A -85,B 0,C 180,E1 -6353.583,E2 -6353.583} C_VEL
LIN {X 0,Y 495.942,Z 320.04,A -85,B 0,C 180,E1 -6353.951,E2 -6353.951} C_VEL
LIN {X 0,Y 495.461,Z 321.812,A -85,B 0,C 180,E1 -6354.6,E2 -6354.6} C_VEL
LIN {X 0,Y 492.748,Z 324.863,A -85,B 0,C 180,E1 -6355.648,E2 -6355.648} C_VEL
LIN {X 0,Y 490.357,Z 327.305,A -85,B 0,C 180,E1 -6356.494,E2 -6356.494} C_VEL
LIN {X 0,Y 489.326,Z 328.96,A -85,B 0,C 180,E1 -6357.152,E2 -6357.152} C_VEL
LIN {X 0,Y 489.247,Z 329.472,A -85,B 0,C 180,E1 -6357.377,E2 -6357.377} C_VEL
LIN {X 0,Y 489.153,Z 334.809,A -85,B 0,C 180,E1 -6359.808,E2 -6359.808} C_VEL
LIN {X 0,Y 489.046,Z 341.379,A -85,B 0,C 180,E1 -6362.999,E2 -6362.999} C_VEL
LIN {X 0,Y 488.915,Z 347.937,A -85,B 0,C 180,E1 -6366.264,E2 -6366.264} C_VEL
LIN {X 0,Y 488.845,Z 353.793,A -85,B 0,C 180,E1 -6369.147,E2 -6369.147} C_VEL
LIN {X 0,Y 488.754,Z 360.932,A -85,B 0,C 180,E1 -6372.422,E2 -6372.422} C_VEL
LIN {X 0,Y 488.842,Z 367.916,A -85,B 0,C 180,E1 -6375.347,E2 -6375.347} C_VEL
LIN {X 0,Y 491.331,Z 377.011,A -85,B 0,C 180,E1 -6375.651,E2 -6375.651} C_VEL
LIN {X 0,Y 491.159,Z 389.493,A -85,B 0,C 180,E1 -6376.078,E2 -6376.078} C_VEL
LIN {X 0,Y 490.883,Z 401.375,A -85,B 0,C 180,E1 -6376.65,E2 -6376.65} C_VEL
LIN {X 0,Y 490.661,Z 412.64,A -85,B 0,C 180,E1 -6377.364,E2 -6377.364} C_VEL
LIN {X 0,Y 490.281,Z 423.25,A -85,B 0,C 180,E1 -6378.212,E2 -6378.212} C_VEL
LIN {X 0,Y 489.878,Z 433.578,A -85,B 0,C 180,E1 -6379.249,E2 -6379.249} C_VEL
LIN {X 0,Y 489.582,Z 441.979,A -85,B 0,C 180,E1 -6380.288,E2 -6380.288} C_VEL
LIN {X 0,Y 489.201,Z 450.163,A -85,B 0,C 180,E1 -6381.53,E2 -6381.53} C_VEL
LIN {X 0,Y 488.922,Z 456.858,A -85,B 0,C 180,E1 -6382.81,E2 -6382.81} C_VEL
LIN {X 0,Y 488.715,Z 462.655,A -85,B 0,C 180,E1 -6384.221,E2 -6384.221} C_VEL
LIN {X 0,Y 488.53,Z 466.539,A -85,B 0,C 180,E1 -6385.46,E2 -6385.46} C_VEL
LIN {X 0,Y 488.447,Z 469.396,A -85,B 0,C 180,E1 -6386.699,E2 -6386.699} C_VEL
LIN {X 0,Y 488.424,Z 470.782,A -85,B 0,C 180,E1 -6387.524,E2 -6387.524} C_VEL
LIN {X 0,Y 488.358,Z 472.357,A -85,B 0,C 180,E1 -6389.173,E2 -6389.173} C_VEL
LIN {X 0,Y 488.344,Z 472.591,A -85,B 0,C 180,E1 -6389.998,E2 -6389.998} C_VEL
LIN {X 0,Y 488.358,Z 472.41,A -85,B 0,C 180,E1 -6390.823,E2 -6390.823} C_VEL
LIN {X 0,Y 488.307,Z 471.853,A -85,B 0,C 180,E1 -6391.647,E2 -6391.647} C_VEL
LIN {X 0,Y 488.55,Z 469.567,A -85,B 0,C 180,E1 -6393.297,E2 -6393.297} C_VEL
LIN {X 0,Y 488.612,Z 466.783,A -85,B 0,C 180,E1 -6394.535,E2 -6394.535} C_VEL
LIN {X 0,Y 488.706,Z 462.996,A -85,B 0,C 180,E1 -6395.775,E2 -6395.775} C_VEL
LIN {X 0,Y 488.834,Z 458.605,A -85,B 0,C 180,E1 -6396.897,E2 -6396.897} C_VEL
LIN {X 0,Y 489.121,Z 451.865,A -85,B 0,C 180,E1 -6398.259,E2 -6398.259} C_VEL
LIN {X 0,Y 489.504,Z 444.118,A -85,B 0,C 180,E1 -6399.501,E2 -6399.501} C_VEL
LIN {X 0,Y 489.796,Z 436.209,A -85,B 0,C 180,E1 -6400.539,E2 -6400.539} C_VEL
LIN {X 0,Y 490.146,Z 426.498,A -85,B 0,C 180,E1 -6401.578,E2 -6401.578} C_VEL
LIN {X 0,Y 490.557,Z 415.472,A -85,B 0,C 180,E1 -6402.517,E2 -6402.517} C_VEL
LIN {X 0,Y 490.78,Z 404.829,A -85,B 0,C 180,E1 -6403.243,E2 -6403.243} C_VEL
LIN {X 0,Y 491.094,Z 392.869,A -85,B 0,C 180,E1 -6403.867,E2 -6403.867} C_VEL
LIN {X 0,Y 491.3,Z 379.621,A -85,B 0,C 180,E1 -6404.363,E2 -6404.363} C_VEL
LIN {X 0,Y 491.003,Z 375.591,A -85,B 0,C 180,E1 -6404.487,E2 -6404.487} C_VEL
LIN {X 0,Y 488.849,Z 367.9,A -85,B 0,C 180,E1 -6404.756,E2 -6404.756} C_VEL
LIN {X 0,Y 488.748,Z 361.169,A -85,B 0,C 180,E1 -6407.574,E2 -6407.574} C_VEL
LIN {X 0,Y 488.833,Z 353.999,A -85,B 0,C 180,E1 -6410.85,E2 -6410.85} C_VEL
LIN {X 0,Y 488.918,Z 348.135,A -85,B 0,C 180,E1 -6413.731,E2 -6413.731} C_VEL
LIN {X 0,Y 489.008,Z 342.676,A -85,B 0,C 180,E1 -6416.454,E2 -6416.454} C_VEL
LIN {X 0,Y 489.173,Z 336.041,A -85,B 0,C 180,E1 -6419.711,E2 -6419.711} C_VEL
LIN {X 0,Y 489.258,Z 329.818,A -85,B 0,C 180,E1 -6422.59,E2 -6422.59} C_VEL
LIN {X 0,Y 489.267,Z 323.99,A -85,B 0,C 180,E1 -6425.066,E2 -6425.066} C_VEL
LIN {X 0,Y 488.733,Z 319.924,A -85,B 0,C 180,E1 -6426.733,E2 -6426.733} C_VEL
LIN {X 0,Y 488.689,Z 319.925,A -85,B 0,C 180,E1 -6429.252,E2 -6429.252} C_VEL
LIN {X 0,Y 488.674,Z 319.926,A -85,B 0,C 180,E1 -6432.524,E2 -6432.524} C_VEL
LIN {X 0,Y 488.697,Z 319.928,A -85,B 0,C 180,E1 -6435.196,E2 -6435.196} C_VEL
LIN {X 0,Y 488.717,Z 319.919,A -85,B 0,C 180,E1 -6437.477,E2 -6437.477} C_VEL
LIN {X 0,Y 488.737,Z 319.919,A -85,B 0,C 180,E1 -6440.749,E2 -6440.749} C_VEL
LIN {X 0,Y 488.666,Z 319.929,A -85,B 0,C 180,E1 -6443.867,E2 -6443.867} C_VEL
LIN {X 0,Y 488.719,Z 319.919,A -85,B 0,C 180,E1 -6446.875,E2 -6446.875} C_VEL
LIN {X 0,Y 488.703,Z 319.918,A -85,B 0,C 180,E1 -6449.779,E2 -6449.779} C_VEL
LIN {X 0,Y 488.778,Z 319.909,A -85,B 0,C 180,E1 -6453.053,E2 -6453.053} C_VEL
LIN {X 0,Y 488.695,Z 319.923,A -85,B 0,C 180,E1 -6456.254,E2 -6456.254} C_VEL
LIN {X 0,Y 488.725,Z 319.919,A -85,B 0,C 180,E1 -6459.174,E2 -6459.174} C_VEL
LIN {X 0,Y 488.709,Z 319.918,A -85,B 0,C 180,E1 -6462.422,E2 -6462.422} C_VEL
LIN {X 0,Y 488.737,Z 319.916,A -85,B 0,C 180,E1 -6464.999,E2 -6464.999} C_VEL
LIN {X 0,Y 488.815,Z 319.912,A -85,B 0,C 180,E1 -6468.387,E2 -6468.387} C_VEL
LIN {X 0,Y 488.801,Z 319.909,A -85,B 0,C 180,E1 -6471.733,E2 -6471.733} C_VEL
LIN {X 0,Y 488.838,Z 319.902,A -85,B 0,C 180,E1 -6474.224,E2 -6474.224} C_VEL
LIN {X 0,Y 488.931,Z 319.894,A -85,B 0,C 180,E1 -6477.528,E2 -6477.528} C_VEL
LIN {X 0,Y 488.953,Z 319.888,A -85,B 0,C 180,E1 -6480.823,E2 -6480.823} C_VEL
LIN {X 0,Y 488.794,Z 319.909,A -85,B 0,C 180,E1 -6483.297,E2 -6483.297} C_VEL
LIN {X 0,Y 488.852,Z 319.907,A -85,B 0,C 180,E1 -6485.775,E2 -6485.775} C_VEL
LIN {X 0,Y 488.794,Z 319.909,A -85,B 0,C 180,E1 -6488.266,E2 -6488.266} C_VEL
LIN {X 0,Y 488.809,Z 319.909,A -85,B 0,C 180,E1 -6491.612,E2 -6491.612} C_VEL
LIN {X 0,Y 488.738,Z 319.918,A -85,B 0,C 180,E1 -6495.001,E2 -6495.001} C_VEL
LIN {X 0,Y 488.742,Z 319.918,A -85,B 0,C 180,E1 -6498.442,E2 -6498.442} C_VEL
LIN {X 0,Y 488.718,Z 319.92,A -85,B 0,C 180,E1 -6501.07,E2 -6501.07} C_VEL
LIN {X 0,Y 488.687,Z 319.924,A -85,B 0,C 180,E1 -6503.745,E2 -6503.745} C_VEL
LIN {X 0,Y 488.767,Z 319.917,A -85,B 0,C 180,E1 -6506.945,E2 -6506.945} C_VEL
LIN {X 0,Y 488.687,Z 319.927,A -85,B 0,C 180,E1 -6510.364,E2 -6510.364} C_VEL
LIN {X 0,Y 488.714,Z 319.922,A -85,B 0,C 180,E1 -6513.486,E2 -6513.486} C_VEL
LIN {X 0,Y 488.67,Z 319.926,A -85,B 0,C 180,E1 -6516.358,E2 -6516.358} C_VEL
LIN {X 0,Y 488.681,Z 319.927,A -85,B 0,C 180,E1 -6519.256,E2 -6519.256} C_VEL
